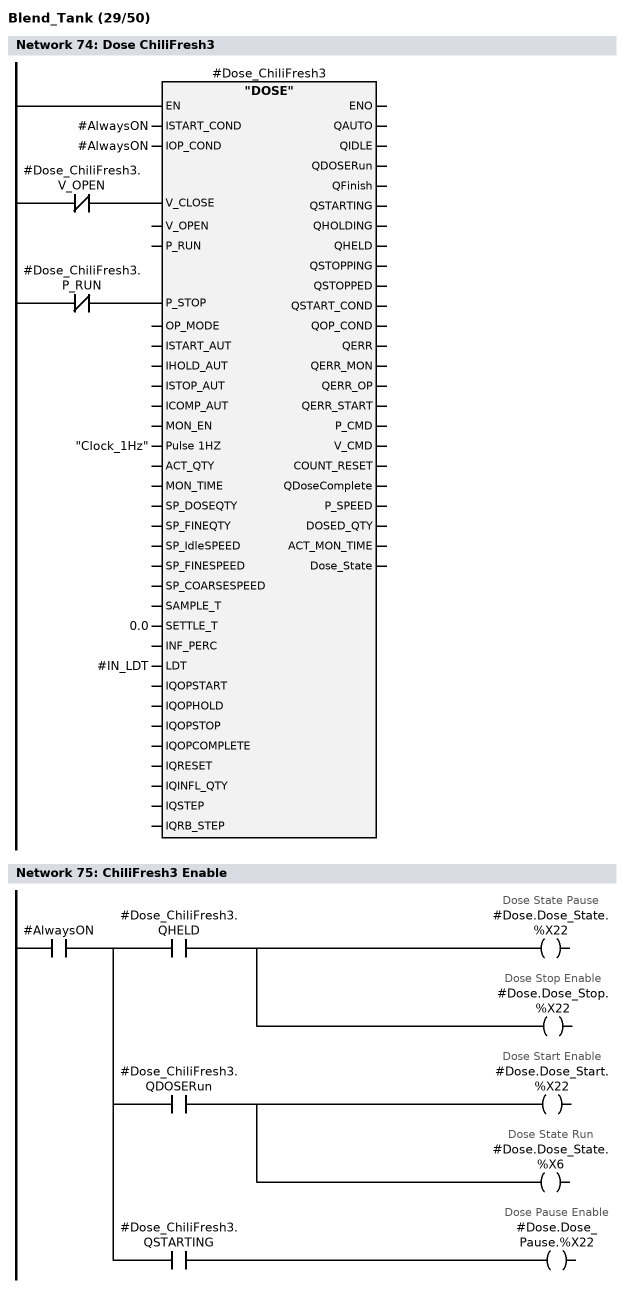
   RUNG wire#powerrail
      #Dose_ChiliFresh3(V_CLOSE := wire#w1, P_STOP := wire#w2, ISTART_COND := #AlwaysON, IOP_COND := #AlwaysON, V_OPEN :=, P_RUN :=, OP_MODE :=, ISTART_AUT :=, IHOLD_AUT :=, ISTOP_AUT :=, ICOMP_AUT :=, MON_EN :=, "Pulse 1HZ" := "Clock_1Hz", ACT_QTY :=, MON_TIME :=, SP_DOSEQTY :=, SP_FINEQTY :=, SP_IdleSPEED :=, SP_FINESPEED :=, SP_COARSESPEED :=, SAMPLE_T :=, SETTLE_T := 0.0, INF_PERC :=, LDT := #IN_LDT, IQOPSTART :=, IQOPHOLD :=, IQOPSTOP :=, IQOPCOMPLETE :=, IQRESET :=, IQINFL_QTY :=, IQSTEP :=, IQRB_STEP :=, QAUTO =>, QIDLE =>, QDOSERun =>, QFinish =>, QSTARTING =>, QHOLDING =>, QHELD =>, QSTOPPING =>, QSTOPPED =>, QSTART_COND =>, QOP_COND =>, QERR =>, QERR_MON =>, QERR_OP =>, QERR_START =>, P_CMD =>, V_CMD =>, COUNT_RESET =>, QDoseComplete =>, P_SPEED =>, DOSED_QTY =>, ACT_MON_TIME =>, Dose_State =>)
   END_RUNG
   RUNG wire#powerrail
      I_Contact( #Dose_ChiliFresh3.V_OPEN )
   END_RUNG wire#w1
   RUNG wire#powerrail
      I_Contact( #Dose_ChiliFresh3.P_RUN )
   END_RUNG wire#w2
   // the same network as SCL:
   #Dose_ChiliFresh3(ISTART_COND := #AlwaysON,   // "DOSE"
                     IOP_COND := #AlwaysON,
                     V_CLOSE := NOT #Dose_ChiliFresh3.V_OPEN,
                     P_STOP := NOT #Dose_ChiliFresh3.P_RUN,
                     "Pulse 1HZ" := "Clock_1Hz",
                     SETTLE_T := 0.0,
                     LDT := #IN_LDT);
END_REGION

REGION Network 75: ChiliFresh3 Enable
   RUNG wire#powerrail
      Contact( #AlwaysON )
      wire#w1
      Contact( #Dose_ChiliFresh3.QHELD )
      wire#w2
      Coil( #Dose.Dose_State.%X22 )   // Dose State Pause
   END_RUNG
   RUNG wire#w2
      Coil( #Dose.Dose_Stop.%X22 )   // Dose Stop Enable
   END_RUNG
   RUNG wire#w1
      Contact( #Dose_ChiliFresh3.QDOSERun )
      wire#w3
      Coil( #Dose.Dose_Start.%X22 )   // Dose Start Enable
   END_RUNG
   RUNG wire#w3
      Coil( #Dose.Dose_State.%X6 )   // Dose State Run
   END_RUNG
   RUNG wire#w1
      Contact( #Dose_ChiliFresh3.QSTARTING )
      Coil( #Dose.Dose_Pause.%X22 )   // Dose Pause Enable
   END_RUNG
   // the same network as SCL:
   #Dose.Dose_State.%X22 := #AlwaysON AND #Dose_ChiliFresh3.QHELD;   // Dose State Pause
   #Dose.Dose_Stop.%X22 := #Dose.Dose_State.%X22;   // Dose Stop Enable
   #Dose.Dose_Start.%X22 := #AlwaysON AND #Dose_ChiliFresh3.QDOSERun;   // Dose Start Enable
   #Dose.Dose_State.%X6 := #Dose.Dose_Start.%X22;   // Dose State Run
   #Dose.Dose_Pause.%X22 := #AlwaysON AND #Dose_ChiliFresh3.QSTARTING;   // Dose Pause Enable
END_REGION

REGION Network 76: ChiliFresh3 Header Req
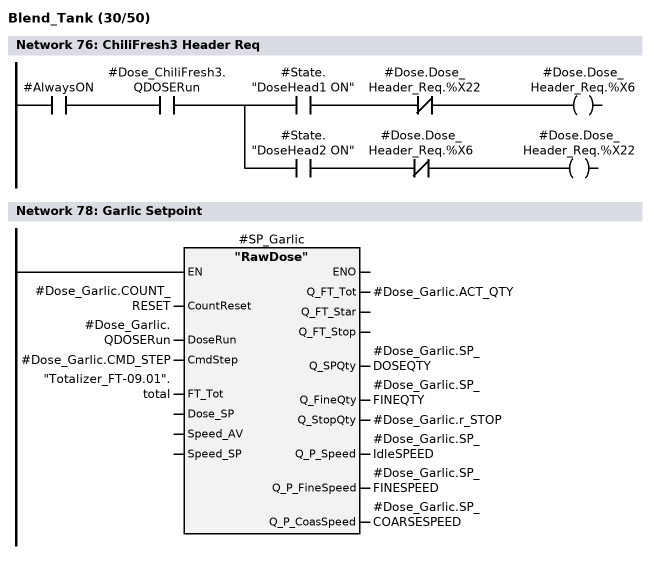
   RUNG wire#powerrail
      Contact( #AlwaysON )
      Contact( #Dose_ChiliFresh3.QDOSERun )
      wire#w1
      Contact( #State."DoseHead1 ON" )
      I_Contact( #Dose.Dose_Header_Req.%X22 )
      Coil( #Dose.Dose_Header_Req.%X6 )
   END_RUNG
   RUNG wire#w1
      Contact( #State."DoseHead2 ON" )
      I_Contact( #Dose.Dose_Header_Req.%X6 )
      Coil( #Dose.Dose_Header_Req.%X22 )
   END_RUNG
   // the same network as SCL:
   #_w1 := #AlwaysON AND #Dose_ChiliFresh3.QDOSERun;
   #Dose.Dose_Header_Req.%X6 := #_w1 AND #State."DoseHead1 ON" AND NOT #Dose.Dose_Header_Req.%X22;
   #Dose.Dose_Header_Req.%X22 := #_w1 AND #State."DoseHead2 ON" AND NOT #Dose.Dose_Header_Req.%X6;
END_REGION

REGION Network 78: Garlic Setpoint
   RUNG wire#powerrail
      #SP_Garlic(CountReset := #Dose_Garlic.COUNT_RESET, DoseRun := #Dose_Garlic.QDOSERun, CmdStep := #Dose_Garlic.CMD_STEP, FT_Tot := "Totalizer_FT-09.01".total, Dose_SP :=, Speed_AV :=, Speed_SP :=, Q_FT_Tot => #Dose_Garlic.ACT_QTY, Q_FT_Star =>, Q_FT_Stop =>, Q_SPQty => #Dose_Garlic.SP_DOSEQTY, Q_FineQty => #Dose_Garlic.SP_FINEQTY, Q_StopQty => #Dose_Garlic.r_STOP, Q_P_Speed => #Dose_Garlic.SP_IdleSPEED, Q_P_FineSpeed => #Dose_Garlic.SP_FINESPEED, Q_P_CoasSpeed => #Dose_Garlic.SP_COARSESPEED)
   END_RUNG
   // the same network as SCL:
   #SP_Garlic(CountReset := #Dose_Garlic.COUNT_RESET,   // "RawDose"
              DoseRun := #Dose_Garlic.QDOSERun,
              CmdStep := #Dose_Garlic.CMD_STEP,
              FT_Tot := "Totalizer_FT-09.01".total,
              Q_FT_Tot => #Dose_Garlic.ACT_QTY,
              Q_SPQty => #Dose_Garlic.SP_DOSEQTY,
              Q_FineQty => #Dose_Garlic.SP_FINEQTY,
              Q_StopQty => #Dose_Garlic.r_STOP,
              Q_P_Speed => #Dose_Garlic.SP_IdleSPEED,
              Q_P_FineSpeed => #Dose_Garlic.SP_FINESPEED,
              Q_P_CoasSpeed => #Dose_Garlic.SP_COARSESPEED);
END_REGION

REGION Network 79: Command Dose Garlic
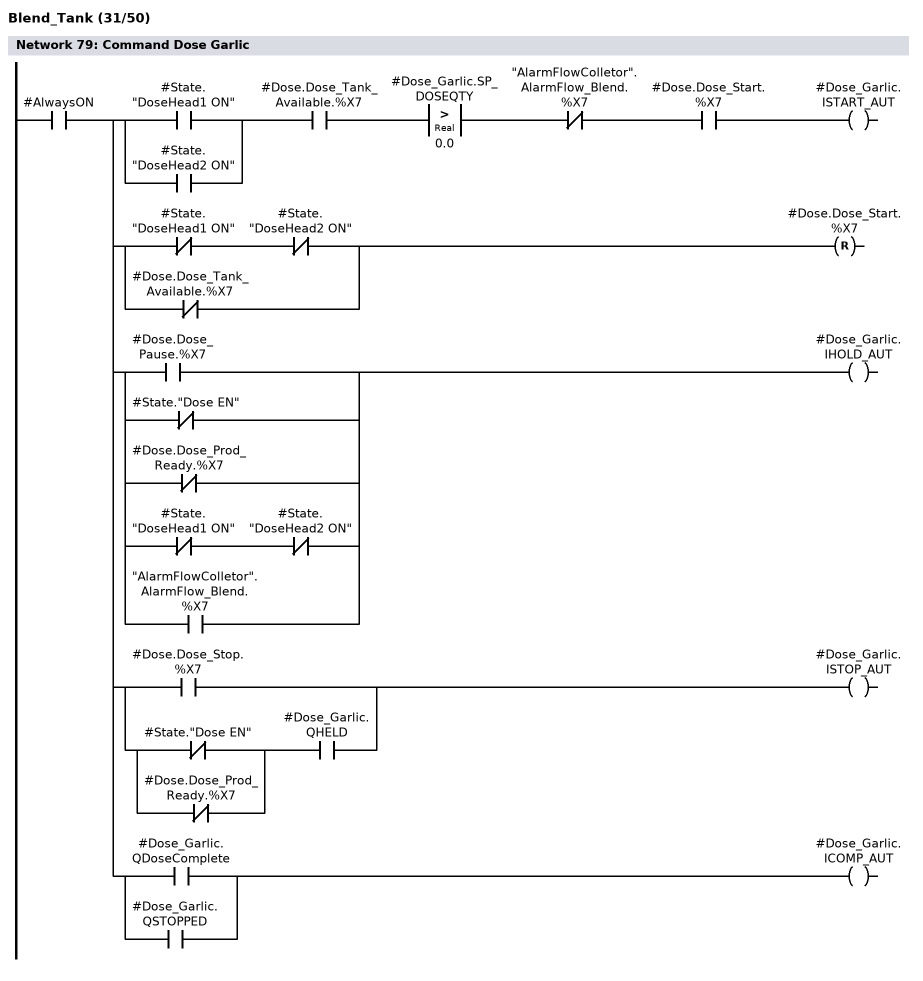
   RUNG wire#powerrail
      Contact( #AlwaysON )
      wire#w1
      Contact( #State."DoseHead1 ON" )
      wire#w2
      Contact( #Dose.Dose_Tank_Available.%X7 )
      { S7_Templates := "SrcType := Real" } GT_Contact(in1 := #Dose_Garlic.SP_DOSEQTY, in2 := 0.0)
      I_Contact( "AlarmFlowColletor".AlarmFlow_Blend.%X7 )
      Contact( #Dose.Dose_Start.%X7 )
      Coil( #Dose_Garlic.ISTART_AUT )
   END_RUNG
   RUNG wire#w1
      Contact( #State."DoseHead2 ON" )
   END_RUNG wire#w2
   RUNG wire#w1
      I_Contact( #State."DoseHead1 ON" )
      I_Contact( #State."DoseHead2 ON" )
      wire#w3
      R_Coil( #Dose.Dose_Start.%X7 )
   END_RUNG
   RUNG wire#w1
      I_Contact( #Dose.Dose_Tank_Available.%X7 )
   END_RUNG wire#w3
   RUNG wire#w1
      Contact( #Dose.Dose_Pause.%X7 )
      wire#w4
      Coil( #Dose_Garlic.IHOLD_AUT )
   END_RUNG
   RUNG wire#w1
      I_Contact( #State."Dose EN" )
   END_RUNG wire#w4
   RUNG wire#w1
      I_Contact( #Dose.Dose_Prod_Ready.%X7 )
   END_RUNG wire#w4
   RUNG wire#w1
      I_Contact( #State."DoseHead1 ON" )
      I_Contact( #State."DoseHead2 ON" )
   END_RUNG wire#w4
   RUNG wire#w1
      Contact( "AlarmFlowColletor".AlarmFlow_Blend.%X7 )
   END_RUNG wire#w4
   RUNG wire#w1
      Contact( #Dose.Dose_Stop.%X7 )
      wire#w5
      Coil( #Dose_Garlic.ISTOP_AUT )
   END_RUNG
   RUNG wire#w1
      I_Contact( #State."Dose EN" )
      wire#w6
      Contact( #Dose_Garlic.QHELD )
   END_RUNG wire#w5
   RUNG wire#w1
      I_Contact( #Dose.Dose_Prod_Ready.%X7 )
   END_RUNG wire#w6
   RUNG wire#w1
      Contact( #Dose_Garlic.QDoseComplete )
      wire#w7
      Coil( #Dose_Garlic.ICOMP_AUT )
   END_RUNG
   RUNG wire#w1
      Contact( #Dose_Garlic.QSTOPPED )
   END_RUNG wire#w7
   // the same network as SCL:
   #Dose_Garlic.ISTART_AUT := #AlwaysON AND (#State."DoseHead1 ON" OR #State."DoseHead2 ON") AND #Dose.Dose_Tank_Available.%X7 AND (#Dose_Garlic.SP_DOSEQTY > 0.0) AND NOT "AlarmFlowColletor".AlarmFlow_Blend.%X7 AND #Dose.Dose_Start.%X7;
   IF #AlwaysON AND ((NOT #State."DoseHead1 ON" AND NOT #State."DoseHead2 ON") OR NOT #Dose.Dose_Tank_Available.%X7) THEN
       #Dose.Dose_Start.%X7 := FALSE;
   END_IF;
   #Dose_Garlic.IHOLD_AUT := #AlwaysON AND (#Dose.Dose_Pause.%X7 OR NOT #State."Dose EN" OR NOT #Dose.Dose_Prod_Ready.%X7 OR (NOT #State."DoseHead1 ON" AND NOT #State."DoseHead2 ON") OR "AlarmFlowColletor".AlarmFlow_Blend.%X7);
   #Dose_Garlic.ISTOP_AUT := #AlwaysON AND (#Dose.Dose_Stop.%X7 OR ((NOT #State."Dose EN" OR NOT #Dose.Dose_Prod_Ready.%X7) AND #Dose_Garlic.QHELD));
   #Dose_Garlic.ICOMP_AUT := #AlwaysON AND (#Dose_Garlic.QDoseComplete OR #Dose_Garlic.QSTOPPED);
END_REGION

REGION Network 80: Dose Garlic
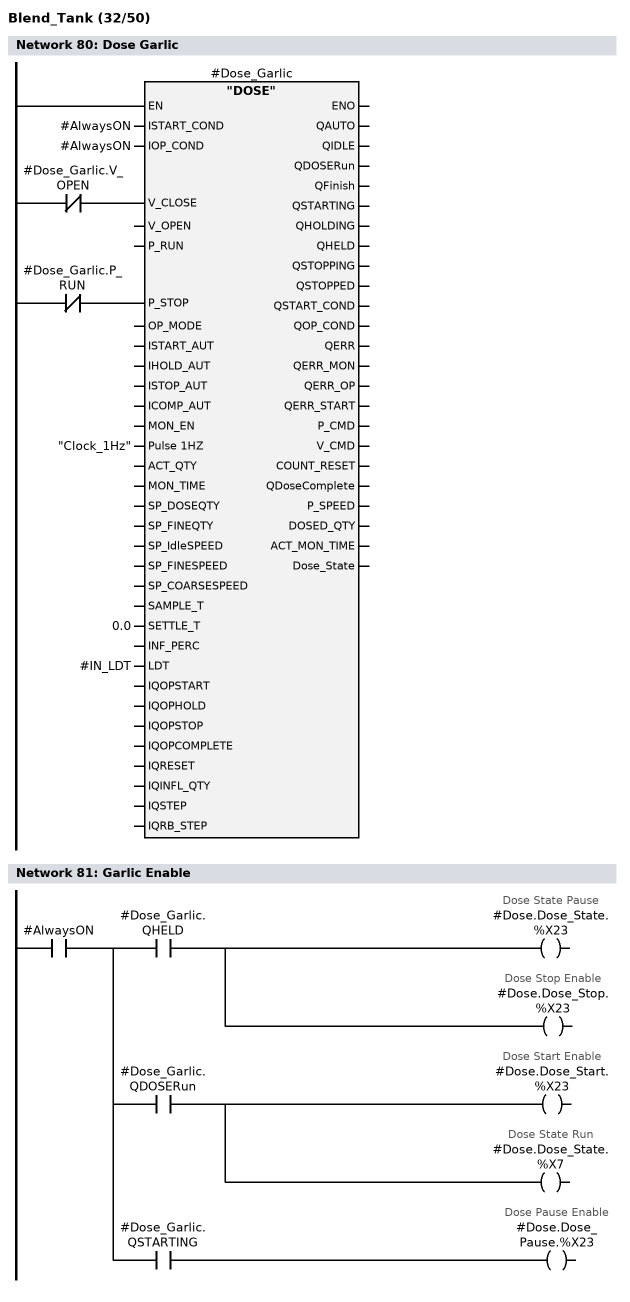
   RUNG wire#powerrail
      #Dose_Garlic(V_CLOSE := wire#w1, P_STOP := wire#w2, ISTART_COND := #AlwaysON, IOP_COND := #AlwaysON, V_OPEN :=, P_RUN :=, OP_MODE :=, ISTART_AUT :=, IHOLD_AUT :=, ISTOP_AUT :=, ICOMP_AUT :=, MON_EN :=, "Pulse 1HZ" := "Clock_1Hz", ACT_QTY :=, MON_TIME :=, SP_DOSEQTY :=, SP_FINEQTY :=, SP_IdleSPEED :=, SP_FINESPEED :=, SP_COARSESPEED :=, SAMPLE_T :=, SETTLE_T := 0.0, INF_PERC :=, LDT := #IN_LDT, IQOPSTART :=, IQOPHOLD :=, IQOPSTOP :=, IQOPCOMPLETE :=, IQRESET :=, IQINFL_QTY :=, IQSTEP :=, IQRB_STEP :=, QAUTO =>, QIDLE =>, QDOSERun =>, QFinish =>, QSTARTING =>, QHOLDING =>, QHELD =>, QSTOPPING =>, QSTOPPED =>, QSTART_COND =>, QOP_COND =>, QERR =>, QERR_MON =>, QERR_OP =>, QERR_START =>, P_CMD =>, V_CMD =>, COUNT_RESET =>, QDoseComplete =>, P_SPEED =>, DOSED_QTY =>, ACT_MON_TIME =>, Dose_State =>)
   END_RUNG
   RUNG wire#powerrail
      I_Contact( #Dose_Garlic.V_OPEN )
   END_RUNG wire#w1
   RUNG wire#powerrail
      I_Contact( #Dose_Garlic.P_RUN )
   END_RUNG wire#w2
   // the same network as SCL:
   #Dose_Garlic(ISTART_COND := #AlwaysON,   // "DOSE"
                IOP_COND := #AlwaysON,
                V_CLOSE := NOT #Dose_Garlic.V_OPEN,
                P_STOP := NOT #Dose_Garlic.P_RUN,
                "Pulse 1HZ" := "Clock_1Hz",
                SETTLE_T := 0.0,
                LDT := #IN_LDT);
END_REGION

REGION Network 81: Garlic Enable
   RUNG wire#powerrail
      Contact( #AlwaysON )
      wire#w1
      Contact( #Dose_Garlic.QHELD )
      wire#w2
      Coil( #Dose.Dose_State.%X23 )   // Dose State Pause
   END_RUNG
   RUNG wire#w2
      Coil( #Dose.Dose_Stop.%X23 )   // Dose Stop Enable
   END_RUNG
   RUNG wire#w1
      Contact( #Dose_Garlic.QDOSERun )
      wire#w3
      Coil( #Dose.Dose_Start.%X23 )   // Dose Start Enable
   END_RUNG
   RUNG wire#w3
      Coil( #Dose.Dose_State.%X7 )   // Dose State Run
   END_RUNG
   RUNG wire#w1
      Contact( #Dose_Garlic.QSTARTING )
      Coil( #Dose.Dose_Pause.%X23 )   // Dose Pause Enable
   END_RUNG
   // the same network as SCL:
   #Dose.Dose_State.%X23 := #AlwaysON AND #Dose_Garlic.QHELD;   // Dose State Pause
   #Dose.Dose_Stop.%X23 := #Dose.Dose_State.%X23;   // Dose Stop Enable
   #Dose.Dose_Start.%X23 := #AlwaysON AND #Dose_Garlic.QDOSERun;   // Dose Start Enable
   #Dose.Dose_State.%X7 := #Dose.Dose_Start.%X23;   // Dose State Run
   #Dose.Dose_Pause.%X23 := #AlwaysON AND #Dose_Garlic.QSTARTING;   // Dose Pause Enable
END_REGION

REGION Network 82: Garlic Header Req
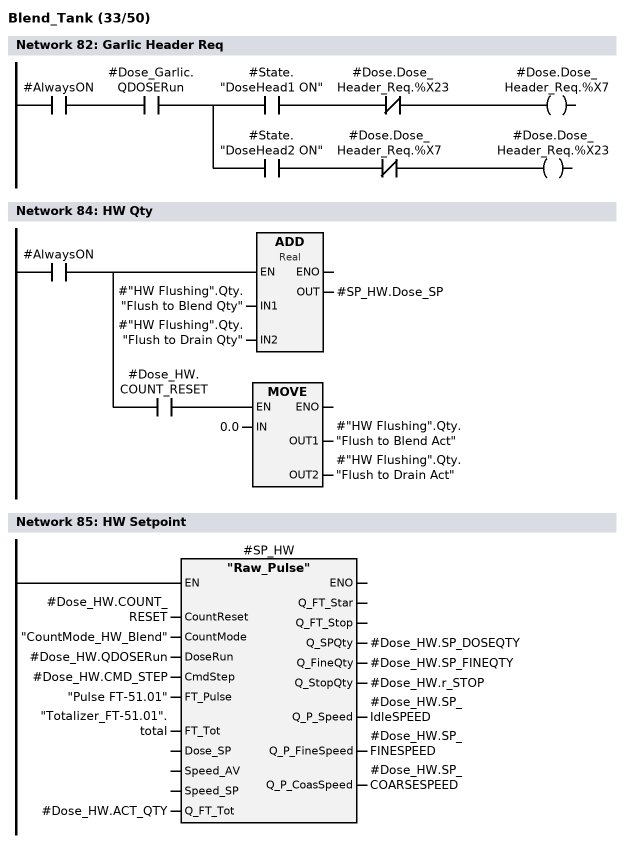
   RUNG wire#powerrail
      Contact( #AlwaysON )
      Contact( #Dose_Garlic.QDOSERun )
      wire#w1
      Contact( #State."DoseHead1 ON" )
      I_Contact( #Dose.Dose_Header_Req.%X23 )
      Coil( #Dose.Dose_Header_Req.%X7 )
   END_RUNG
   RUNG wire#w1
      Contact( #State."DoseHead2 ON" )
      I_Contact( #Dose.Dose_Header_Req.%X7 )
      Coil( #Dose.Dose_Header_Req.%X23 )
   END_RUNG
   // the same network as SCL:
   #_w1 := #AlwaysON AND #Dose_Garlic.QDOSERun;
   #Dose.Dose_Header_Req.%X7 := #_w1 AND #State."DoseHead1 ON" AND NOT #Dose.Dose_Header_Req.%X23;
   #Dose.Dose_Header_Req.%X23 := #_w1 AND #State."DoseHead2 ON" AND NOT #Dose.Dose_Header_Req.%X7;
END_REGION

REGION Network 84: HW Qty
   RUNG wire#powerrail
      Contact( #AlwaysON )
      wire#w1
      { S7_Templates := "SrcType := Real" } Add(in1 := #"HW Flushing".Qty."Flush to Blend Qty", in2 := #"HW Flushing".Qty."Flush to Drain Qty", out => #SP_HW.Dose_SP)
   END_RUNG
   RUNG wire#w1
      Contact( #Dose_HW.COUNT_RESET )
      Move(in := 0.0, out1 => #"HW Flushing".Qty."Flush to Blend Act", out2 => #"HW Flushing".Qty."Flush to Drain Act")
   END_RUNG
   // the same network as SCL:
   IF #AlwaysON THEN
       #SP_HW.Dose_SP := #"HW Flushing".Qty."Flush to Blend Qty" + #"HW Flushing".Qty."Flush to Drain Qty";
   END_IF;
   IF #AlwaysON AND #Dose_HW.COUNT_RESET THEN
       #"HW Flushing".Qty."Flush to Blend Act" := 0.0;
       #"HW Flushing".Qty."Flush to Drain Act" := 0.0;
   END_IF;
END_REGION

REGION Network 85: HW Setpoint
   RUNG wire#powerrail
      #SP_HW(CountReset := #Dose_HW.COUNT_RESET, CountMode := "CountMode_HW_Blend", DoseRun := #Dose_HW.QDOSERun, CmdStep := #Dose_HW.CMD_STEP, FT_Pulse := "Pulse FT-51.01", FT_Tot := "Totalizer_FT-51.01".total, Dose_SP :=, Speed_AV :=, Speed_SP :=, Q_FT_Tot := #Dose_HW.ACT_QTY, Q_FT_Star =>, Q_FT_Stop =>, Q_SPQty => #Dose_HW.SP_DOSEQTY, Q_FineQty => #Dose_HW.SP_FINEQTY, Q_StopQty => #Dose_HW.r_STOP, Q_P_Speed => #Dose_HW.SP_IdleSPEED, Q_P_FineSpeed => #Dose_HW.SP_FINESPEED, Q_P_CoasSpeed => #Dose_HW.SP_COARSESPEED)
   END_RUNG
   // the same network as SCL:
   #SP_HW(CountReset := #Dose_HW.COUNT_RESET,   // "Raw_Pulse"
          CountMode := "CountMode_HW_Blend",
          DoseRun := #Dose_HW.QDOSERun,
          CmdStep := #Dose_HW.CMD_STEP,
          FT_Pulse := "Pulse FT-51.01",
          FT_Tot := "Totalizer_FT-51.01".total,
          Q_FT_Tot := #Dose_HW.ACT_QTY,
          Q_SPQty => #Dose_HW.SP_DOSEQTY,
          Q_FineQty => #Dose_HW.SP_FINEQTY,
          Q_StopQty => #Dose_HW.r_STOP,
          Q_P_Speed => #Dose_HW.SP_IdleSPEED,
          Q_P_FineSpeed => #Dose_HW.SP_FINESPEED,
          Q_P_CoasSpeed => #Dose_HW.SP_COARSESPEED);
END_REGION

REGION Network 86: Command Dose HW
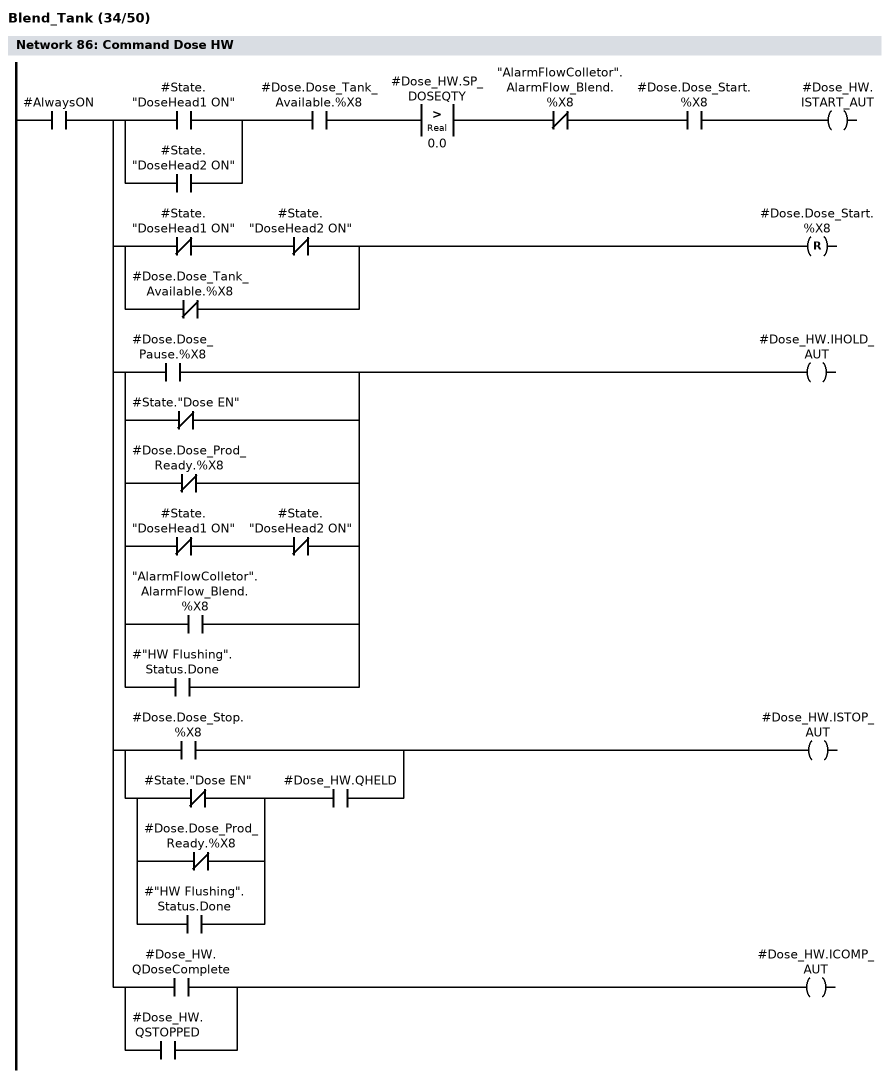
   RUNG wire#powerrail
      Contact( #AlwaysON )
      wire#w1
      Contact( #State."DoseHead1 ON" )
      wire#w2
      Contact( #Dose.Dose_Tank_Available.%X8 )
      { S7_Templates := "SrcType := Real" } GT_Contact(in1 := #Dose_HW.SP_DOSEQTY, in2 := 0.0)
      I_Contact( "AlarmFlowColletor".AlarmFlow_Blend.%X8 )
      Contact( #Dose.Dose_Start.%X8 )
      Coil( #Dose_HW.ISTART_AUT )
   END_RUNG
   RUNG wire#w1
      Contact( #State."DoseHead2 ON" )
   END_RUNG wire#w2
   RUNG wire#w1
      I_Contact( #State."DoseHead1 ON" )
      I_Contact( #State."DoseHead2 ON" )
      wire#w3
      R_Coil( #Dose.Dose_Start.%X8 )
   END_RUNG
   RUNG wire#w1
      I_Contact( #Dose.Dose_Tank_Available.%X8 )
   END_RUNG wire#w3
   RUNG wire#w1
      Contact( #Dose.Dose_Pause.%X8 )
      wire#w4
      Coil( #Dose_HW.IHOLD_AUT )
   END_RUNG
   RUNG wire#w1
      I_Contact( #State."Dose EN" )
   END_RUNG wire#w4
   RUNG wire#w1
      I_Contact( #Dose.Dose_Prod_Ready.%X8 )
   END_RUNG wire#w4
   RUNG wire#w1
      I_Contact( #State."DoseHead1 ON" )
      I_Contact( #State."DoseHead2 ON" )
   END_RUNG wire#w4
   RUNG wire#w1
      Contact( "AlarmFlowColletor".AlarmFlow_Blend.%X8 )
   END_RUNG wire#w4
   RUNG wire#w1
      Contact( #"HW Flushing".Status.Done )
   END_RUNG wire#w4
   RUNG wire#w1
      Contact( #Dose.Dose_Stop.%X8 )
      wire#w5
      Coil( #Dose_HW.ISTOP_AUT )
   END_RUNG
   RUNG wire#w1
      I_Contact( #State."Dose EN" )
      wire#w6
      Contact( #Dose_HW.QHELD )
   END_RUNG wire#w5
   RUNG wire#w1
      I_Contact( #Dose.Dose_Prod_Ready.%X8 )
   END_RUNG wire#w6
   RUNG wire#w1
      Contact( #"HW Flushing".Status.Done )
   END_RUNG wire#w6
   RUNG wire#w1
      Contact( #Dose_HW.QDoseComplete )
      wire#w7
      Coil( #Dose_HW.ICOMP_AUT )
   END_RUNG
   RUNG wire#w1
      Contact( #Dose_HW.QSTOPPED )
   END_RUNG wire#w7
   // the same network as SCL:
   #Dose_HW.ISTART_AUT := #AlwaysON AND (#State."DoseHead1 ON" OR #State."DoseHead2 ON") AND #Dose.Dose_Tank_Available.%X8 AND (#Dose_HW.SP_DOSEQTY > 0.0) AND NOT "AlarmFlowColletor".AlarmFlow_Blend.%X8 AND #Dose.Dose_Start.%X8;
   IF #AlwaysON AND ((NOT #State."DoseHead1 ON" AND NOT #State."DoseHead2 ON") OR NOT #Dose.Dose_Tank_Available.%X8) THEN
       #Dose.Dose_Start.%X8 := FALSE;
   END_IF;
   #Dose_HW.IHOLD_AUT := #AlwaysON AND (#Dose.Dose_Pause.%X8 OR NOT #State."Dose EN" OR NOT #Dose.Dose_Prod_Ready.%X8 OR (NOT #State."DoseHead1 ON" AND NOT #State."DoseHead2 ON") OR "AlarmFlowColletor".AlarmFlow_Blend.%X8 OR #"HW Flushing".Status.Done);
   #Dose_HW.ISTOP_AUT := #AlwaysON AND (#Dose.Dose_Stop.%X8 OR ((NOT #State."Dose EN" OR NOT #Dose.Dose_Prod_Ready.%X8 OR #"HW Flushing".Status.Done) AND #Dose_HW.QHELD));
   #Dose_HW.ICOMP_AUT := #AlwaysON AND (#Dose_HW.QDoseComplete OR #Dose_HW.QSTOPPED);
END_REGION

REGION Network 87: Dose HW
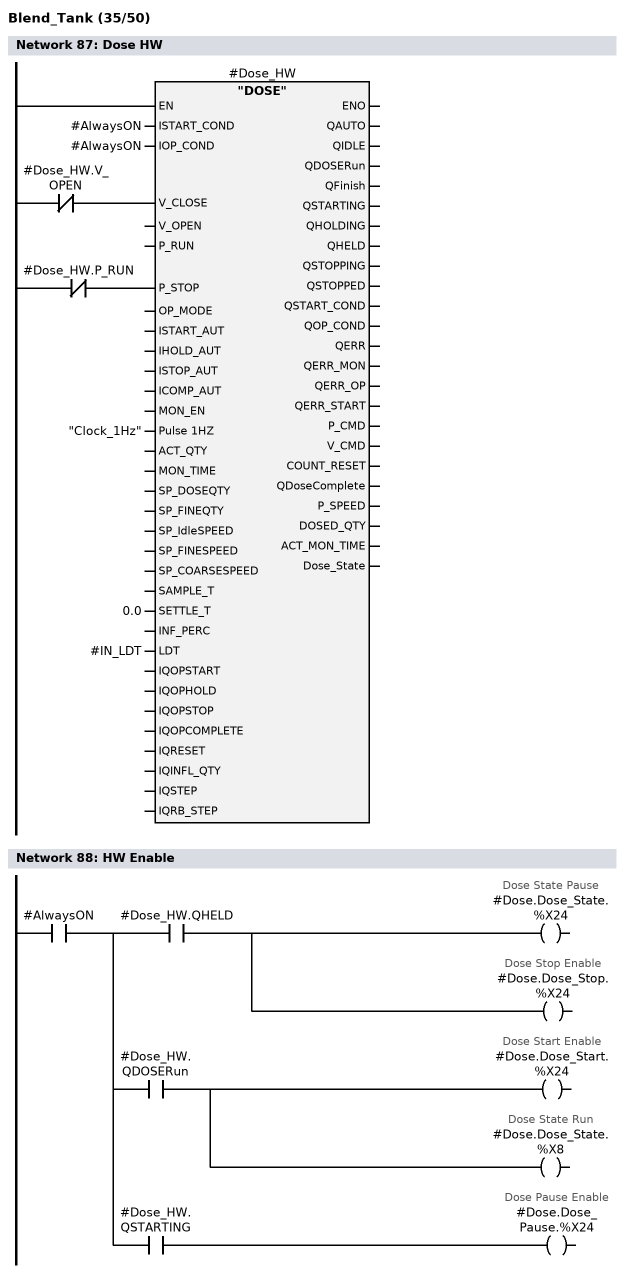
   RUNG wire#powerrail
      #Dose_HW(V_CLOSE := wire#w1, P_STOP := wire#w2, ISTART_COND := #AlwaysON, IOP_COND := #AlwaysON, V_OPEN :=, P_RUN :=, OP_MODE :=, ISTART_AUT :=, IHOLD_AUT :=, ISTOP_AUT :=, ICOMP_AUT :=, MON_EN :=, "Pulse 1HZ" := "Clock_1Hz", ACT_QTY :=, MON_TIME :=, SP_DOSEQTY :=, SP_FINEQTY :=, SP_IdleSPEED :=, SP_FINESPEED :=, SP_COARSESPEED :=, SAMPLE_T :=, SETTLE_T := 0.0, INF_PERC :=, LDT := #IN_LDT, IQOPSTART :=, IQOPHOLD :=, IQOPSTOP :=, IQOPCOMPLETE :=, IQRESET :=, IQINFL_QTY :=, IQSTEP :=, IQRB_STEP :=, QAUTO =>, QIDLE =>, QDOSERun =>, QFinish =>, QSTARTING =>, QHOLDING =>, QHELD =>, QSTOPPING =>, QSTOPPED =>, QSTART_COND =>, QOP_COND =>, QERR =>, QERR_MON =>, QERR_OP =>, QERR_START =>, P_CMD =>, V_CMD =>, COUNT_RESET =>, QDoseComplete =>, P_SPEED =>, DOSED_QTY =>, ACT_MON_TIME =>, Dose_State =>)
   END_RUNG
   RUNG wire#powerrail
      I_Contact( #Dose_HW.V_OPEN )
   END_RUNG wire#w1
   RUNG wire#powerrail
      I_Contact( #Dose_HW.P_RUN )
   END_RUNG wire#w2
   // the same network as SCL:
   #Dose_HW(ISTART_COND := #AlwaysON,   // "DOSE"
            IOP_COND := #AlwaysON,
            V_CLOSE := NOT #Dose_HW.V_OPEN,
            P_STOP := NOT #Dose_HW.P_RUN,
            "Pulse 1HZ" := "Clock_1Hz",
            SETTLE_T := 0.0,
            LDT := #IN_LDT);
END_REGION

REGION Network 88: HW Enable
   RUNG wire#powerrail
      Contact( #AlwaysON )
      wire#w1
      Contact( #Dose_HW.QHELD )
      wire#w2
      Coil( #Dose.Dose_State.%X24 )   // Dose State Pause
   END_RUNG
   RUNG wire#w2
      Coil( #Dose.Dose_Stop.%X24 )   // Dose Stop Enable
   END_RUNG
   RUNG wire#w1
      Contact( #Dose_HW.QDOSERun )
      wire#w3
      Coil( #Dose.Dose_Start.%X24 )   // Dose Start Enable
   END_RUNG
   RUNG wire#w3
      Coil( #Dose.Dose_State.%X8 )   // Dose State Run
   END_RUNG
   RUNG wire#w1
      Contact( #Dose_HW.QSTARTING )
      Coil( #Dose.Dose_Pause.%X24 )   // Dose Pause Enable
   END_RUNG
   // the same network as SCL:
   #Dose.Dose_State.%X24 := #AlwaysON AND #Dose_HW.QHELD;   // Dose State Pause
   #Dose.Dose_Stop.%X24 := #Dose.Dose_State.%X24;   // Dose Stop Enable
   #Dose.Dose_Start.%X24 := #AlwaysON AND #Dose_HW.QDOSERun;   // Dose Start Enable
   #Dose.Dose_State.%X8 := #Dose.Dose_Start.%X24;   // Dose State Run
   #Dose.Dose_Pause.%X24 := #AlwaysON AND #Dose_HW.QSTARTING;   // Dose Pause Enable
END_REGION

REGION Network 89: HW Header Req
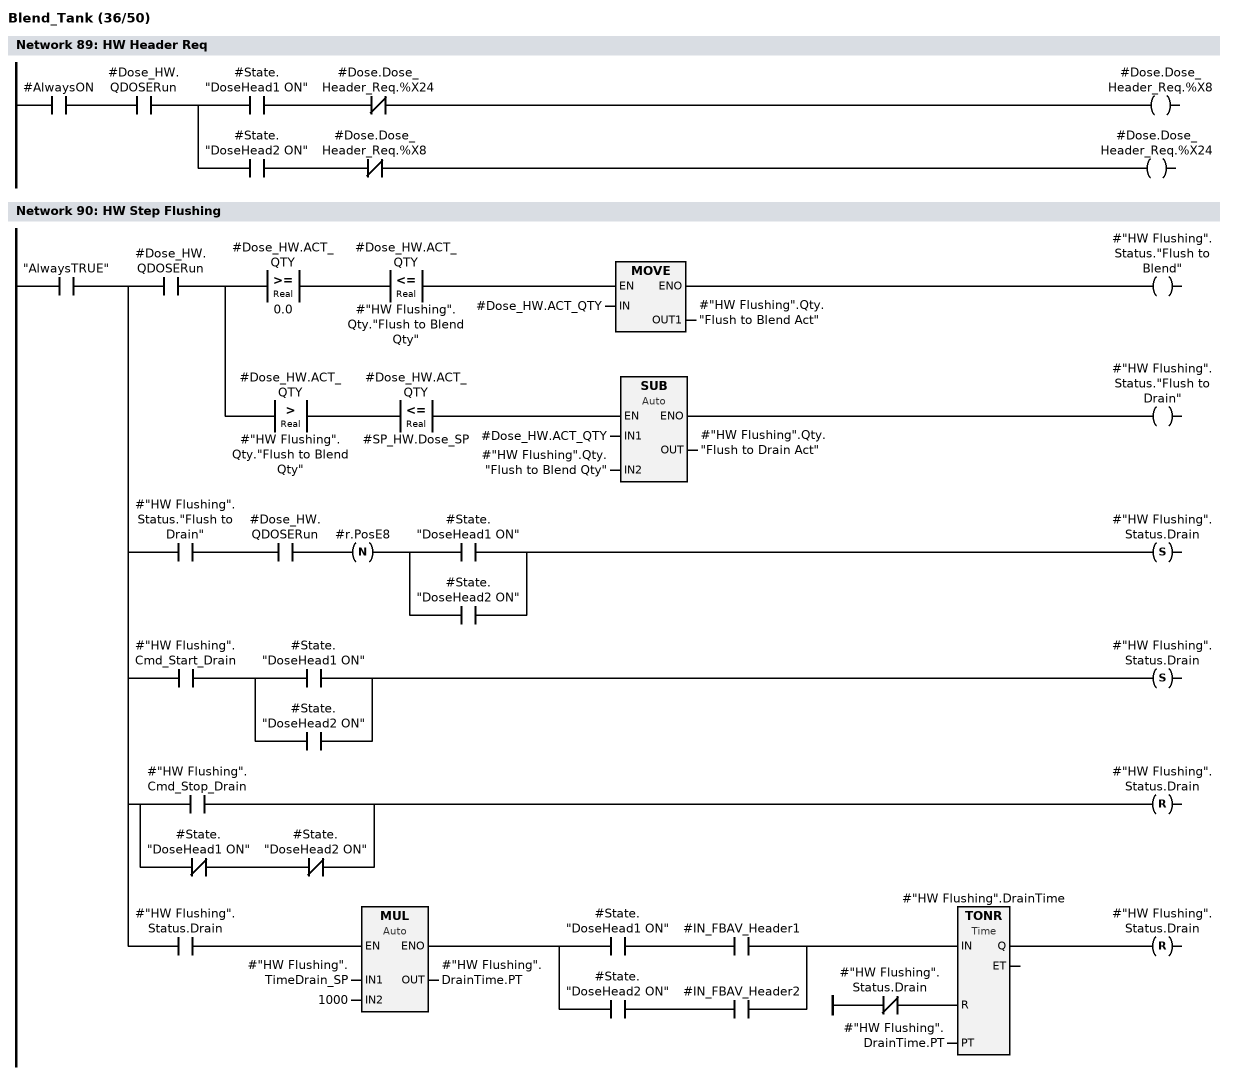
   RUNG wire#powerrail
      Contact( #AlwaysON )
      Contact( #Dose_HW.QDOSERun )
      wire#w1
      Contact( #State."DoseHead1 ON" )
      I_Contact( #Dose.Dose_Header_Req.%X24 )
      Coil( #Dose.Dose_Header_Req.%X8 )
   END_RUNG
   RUNG wire#w1
      Contact( #State."DoseHead2 ON" )
      I_Contact( #Dose.Dose_Header_Req.%X8 )
      Coil( #Dose.Dose_Header_Req.%X24 )
   END_RUNG
   // the same network as SCL:
   #_w1 := #AlwaysON AND #Dose_HW.QDOSERun;
   #Dose.Dose_Header_Req.%X8 := #_w1 AND #State."DoseHead1 ON" AND NOT #Dose.Dose_Header_Req.%X24;
   #Dose.Dose_Header_Req.%X24 := #_w1 AND #State."DoseHead2 ON" AND NOT #Dose.Dose_Header_Req.%X8;
END_REGION

REGION Network 90: HW Step Flushing
   RUNG wire#powerrail
      Contact( "AlwaysTRUE" )
      wire#w1
      Contact( #Dose_HW.QDOSERun )
      wire#w2
      { S7_Templates := "SrcType := Real" } GE_Contact(in1 := #Dose_HW.ACT_QTY, in2 := 0.0)
      { S7_Templates := "SrcType := Real" } LE_Contact(in1 := #Dose_HW.ACT_QTY, in2 := #"HW Flushing".Qty."Flush to Blend Qty")
      Move(in := #Dose_HW.ACT_QTY, out1 => #"HW Flushing".Qty."Flush to Blend Act")
      Coil( #"HW Flushing".Status."Flush to Blend" )
   END_RUNG
   RUNG wire#w2
      { S7_Templates := "SrcType := Real" } GT_Contact(in1 := #Dose_HW.ACT_QTY, in2 := #"HW Flushing".Qty."Flush to Blend Qty")
      { S7_Templates := "SrcType := Real" } LE_Contact(in1 := #Dose_HW.ACT_QTY, in2 := #SP_HW.Dose_SP)
      Sub(in1 := #Dose_HW.ACT_QTY, in2 := #"HW Flushing".Qty."Flush to Blend Qty", out => #"HW Flushing".Qty."Flush to Drain Act")
      Coil( #"HW Flushing".Status."Flush to Drain" )
   END_RUNG
   RUNG wire#w1
      Contact( #"HW Flushing".Status."Flush to Drain" )
      Contact( #Dose_HW.QDOSERun )
      N_Trig( #r.PosE8 )
      wire#w3
      Contact( #State."DoseHead1 ON" )
      wire#w4
      S_Coil( #"HW Flushing".Status.Drain )
   END_RUNG
   RUNG wire#w3
      Contact( #State."DoseHead2 ON" )
   END_RUNG wire#w4
   RUNG wire#w1
      Contact( #"HW Flushing".Cmd_Start_Drain )
      wire#w5
      Contact( #State."DoseHead1 ON" )
      wire#w6
      S_Coil( #"HW Flushing".Status.Drain )
   END_RUNG
   RUNG wire#w5
      Contact( #State."DoseHead2 ON" )
   END_RUNG wire#w6
   RUNG wire#w1
      Contact( #"HW Flushing".Cmd_Stop_Drain )
      wire#w7
      R_Coil( #"HW Flushing".Status.Drain )
   END_RUNG
   RUNG wire#w1
      I_Contact( #State."DoseHead1 ON" )
      I_Contact( #State."DoseHead2 ON" )
   END_RUNG wire#w7
   RUNG wire#w1
      Contact( #"HW Flushing".Status.Drain )
      Mul(in1 := #"HW Flushing".TimeDrain_SP, in2 := 1000, out => #"HW Flushing".DrainTime.PT)
      wire#w8
      Contact( #State."DoseHead1 ON" )
      Contact( #IN_FBAV_Header1 )
      wire#w9
      { S7_Templates := "time_type := Time" } #"HW Flushing".DrainTime.TONR(r := wire#w10, pt := #"HW Flushing".DrainTime.PT, et =>)
      R_Coil( #"HW Flushing".Status.Drain )
   END_RUNG
   RUNG wire#w8
      Contact( #State."DoseHead2 ON" )
      Contact( #IN_FBAV_Header2 )
   END_RUNG wire#w9
   RUNG wire#powerrail
      I_Contact( #"HW Flushing".Status.Drain )
   END_RUNG wire#w10
   // the same network as SCL:
   #_w1 := "AlwaysTRUE" AND #Dose_HW.QDOSERun;
   #_w2 := #_w1 AND (#Dose_HW.ACT_QTY >= 0.0) AND (#Dose_HW.ACT_QTY <= #"HW Flushing".Qty."Flush to Blend Qty");
   IF #_w2 THEN #"HW Flushing".Qty."Flush to Blend Act" := #Dose_HW.ACT_QTY; END_IF;
   #"HW Flushing".Status."Flush to Blend" := #_w2;
   #_w3 := #_w1 AND (#Dose_HW.ACT_QTY > #"HW Flushing".Qty."Flush to Blend Qty") AND (#Dose_HW.ACT_QTY <= #SP_HW.Dose_SP);
   IF #_w3 THEN
       #"HW Flushing".Qty."Flush to Drain Act" := #Dose_HW.ACT_QTY - #"HW Flushing".Qty."Flush to Blend Qty";
   END_IF;
   #"HW Flushing".Status."Flush to Drain" := #_w3;
   #_w4 := "AlwaysTRUE" AND #"HW Flushing".Status."Flush to Drain" AND #Dose_HW.QDOSERun;
   #_w5 := NOT #_w4 AND #r.PosE8;   // falling edge
   #r.PosE8 := #_w4;
   IF #_w5 AND (#State."DoseHead1 ON" OR #State."DoseHead2 ON") THEN
       #"HW Flushing".Status.Drain := TRUE;
   END_IF;
   IF "AlwaysTRUE" AND #"HW Flushing".Cmd_Start_Drain AND (#State."DoseHead1 ON" OR #State."DoseHead2 ON") THEN
       #"HW Flushing".Status.Drain := TRUE;
   END_IF;
   IF "AlwaysTRUE" AND (#"HW Flushing".Cmd_Stop_Drain OR (NOT #State."DoseHead1 ON" AND NOT #State."DoseHead2 ON")) THEN
       #"HW Flushing".Status.Drain := FALSE;
   END_IF;
   #_w6 := "AlwaysTRUE" AND #"HW Flushing".Status.Drain;
   IF #_w6 THEN #"HW Flushing".DrainTime.PT := #"HW Flushing".TimeDrain_SP * 1000; END_IF;
   #"HW Flushing".DrainTime.TONR(IN := #_w6 AND ((#State."DoseHead1 ON" AND #IN_FBAV_Header1) OR (#State."DoseHead2 ON" AND #IN_FBAV_Header2)),
                           R := NOT #"HW Flushing".Status.Drain,
                           PT := #"HW Flushing".DrainTime.PT);
   IF #"HW Flushing".DrainTime.Q THEN #"HW Flushing".Status.Drain := FALSE; END_IF;
END_REGION

REGION Network 92: Vinegar Setpoint
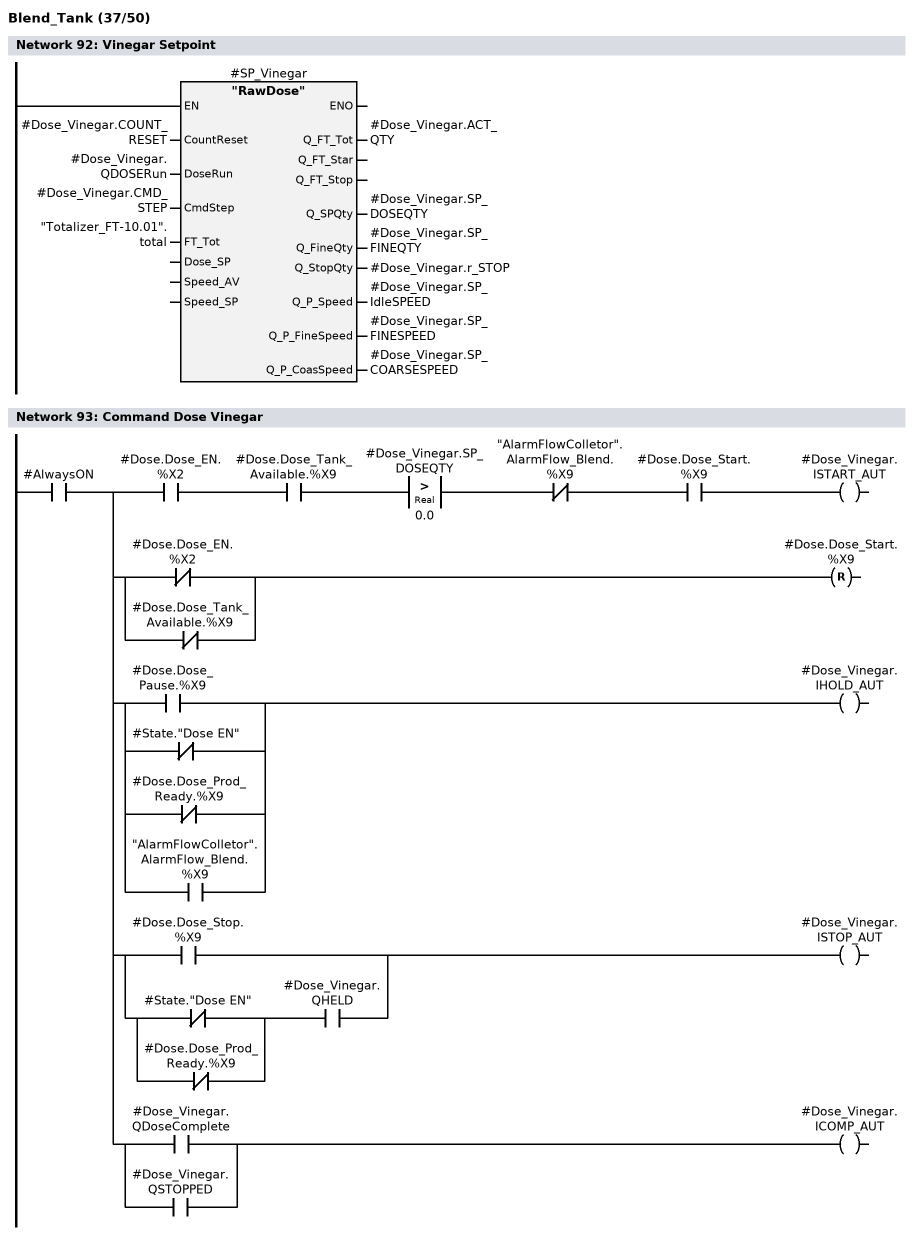
   RUNG wire#powerrail
      #SP_Vinegar(CountReset := #Dose_Vinegar.COUNT_RESET, DoseRun := #Dose_Vinegar.QDOSERun, CmdStep := #Dose_Vinegar.CMD_STEP, FT_Tot := "Totalizer_FT-10.01".total, Dose_SP :=, Speed_AV :=, Speed_SP :=, Q_FT_Tot => #Dose_Vinegar.ACT_QTY, Q_FT_Star =>, Q_FT_Stop =>, Q_SPQty => #Dose_Vinegar.SP_DOSEQTY, Q_FineQty => #Dose_Vinegar.SP_FINEQTY, Q_StopQty => #Dose_Vinegar.r_STOP, Q_P_Speed => #Dose_Vinegar.SP_IdleSPEED, Q_P_FineSpeed => #Dose_Vinegar.SP_FINESPEED, Q_P_CoasSpeed => #Dose_Vinegar.SP_COARSESPEED)
   END_RUNG
   // the same network as SCL:
   #SP_Vinegar(CountReset := #Dose_Vinegar.COUNT_RESET,   // "RawDose"
               DoseRun := #Dose_Vinegar.QDOSERun,
               CmdStep := #Dose_Vinegar.CMD_STEP,
               FT_Tot := "Totalizer_FT-10.01".total,
               Q_FT_Tot => #Dose_Vinegar.ACT_QTY,
               Q_SPQty => #Dose_Vinegar.SP_DOSEQTY,
               Q_FineQty => #Dose_Vinegar.SP_FINEQTY,
               Q_StopQty => #Dose_Vinegar.r_STOP,
               Q_P_Speed => #Dose_Vinegar.SP_IdleSPEED,
               Q_P_FineSpeed => #Dose_Vinegar.SP_FINESPEED,
               Q_P_CoasSpeed => #Dose_Vinegar.SP_COARSESPEED);
END_REGION

REGION Network 93: Command Dose Vinegar
   RUNG wire#powerrail
      Contact( #AlwaysON )
      wire#w1
      Contact( #Dose.Dose_EN.%X2 )
      Contact( #Dose.Dose_Tank_Available.%X9 )
      { S7_Templates := "SrcType := Real" } GT_Contact(in1 := #Dose_Vinegar.SP_DOSEQTY, in2 := 0.0)
      I_Contact( "AlarmFlowColletor".AlarmFlow_Blend.%X9 )
      Contact( #Dose.Dose_Start.%X9 )
      Coil( #Dose_Vinegar.ISTART_AUT )
   END_RUNG
   RUNG wire#w1
      I_Contact( #Dose.Dose_EN.%X2 )
      wire#w2
      R_Coil( #Dose.Dose_Start.%X9 )
   END_RUNG
   RUNG wire#w1
      I_Contact( #Dose.Dose_Tank_Available.%X9 )
   END_RUNG wire#w2
   RUNG wire#w1
      Contact( #Dose.Dose_Pause.%X9 )
      wire#w3
      Coil( #Dose_Vinegar.IHOLD_AUT )
   END_RUNG
   RUNG wire#w1
      I_Contact( #State."Dose EN" )
   END_RUNG wire#w3
   RUNG wire#w1
      I_Contact( #Dose.Dose_Prod_Ready.%X9 )
   END_RUNG wire#w3
   RUNG wire#w1
      Contact( "AlarmFlowColletor".AlarmFlow_Blend.%X9 )
   END_RUNG wire#w3
   RUNG wire#w1
      Contact( #Dose.Dose_Stop.%X9 )
      wire#w4
      Coil( #Dose_Vinegar.ISTOP_AUT )
   END_RUNG
   RUNG wire#w1
      I_Contact( #State."Dose EN" )
      wire#w5
      Contact( #Dose_Vinegar.QHELD )
   END_RUNG wire#w4
   RUNG wire#w1
      I_Contact( #Dose.Dose_Prod_Ready.%X9 )
   END_RUNG wire#w5
   RUNG wire#w1
      Contact( #Dose_Vinegar.QDoseComplete )
      wire#w6
      Coil( #Dose_Vinegar.ICOMP_AUT )
   END_RUNG
   RUNG wire#w1
      Contact( #Dose_Vinegar.QSTOPPED )
   END_RUNG wire#w6
   // the same network as SCL:
   #Dose_Vinegar.ISTART_AUT := #AlwaysON AND #Dose.Dose_EN.%X2 AND #Dose.Dose_Tank_Available.%X9 AND (#Dose_Vinegar.SP_DOSEQTY > 0.0) AND NOT "AlarmFlowColletor".AlarmFlow_Blend.%X9 AND #Dose.Dose_Start.%X9;
   IF #AlwaysON AND (NOT #Dose.Dose_EN.%X2 OR NOT #Dose.Dose_Tank_Available.%X9) THEN
       #Dose.Dose_Start.%X9 := FALSE;
   END_IF;
   #Dose_Vinegar.IHOLD_AUT := #AlwaysON AND (#Dose.Dose_Pause.%X9 OR NOT #State."Dose EN" OR NOT #Dose.Dose_Prod_Ready.%X9 OR "AlarmFlowColletor".AlarmFlow_Blend.%X9);
   #Dose_Vinegar.ISTOP_AUT := #AlwaysON AND (#Dose.Dose_Stop.%X9 OR ((NOT #State."Dose EN" OR NOT #Dose.Dose_Prod_Ready.%X9) AND #Dose_Vinegar.QHELD));
   #Dose_Vinegar.ICOMP_AUT := #AlwaysON AND (#Dose_Vinegar.QDoseComplete OR #Dose_Vinegar.QSTOPPED);
END_REGION

REGION Network 94: Dose Vinegar
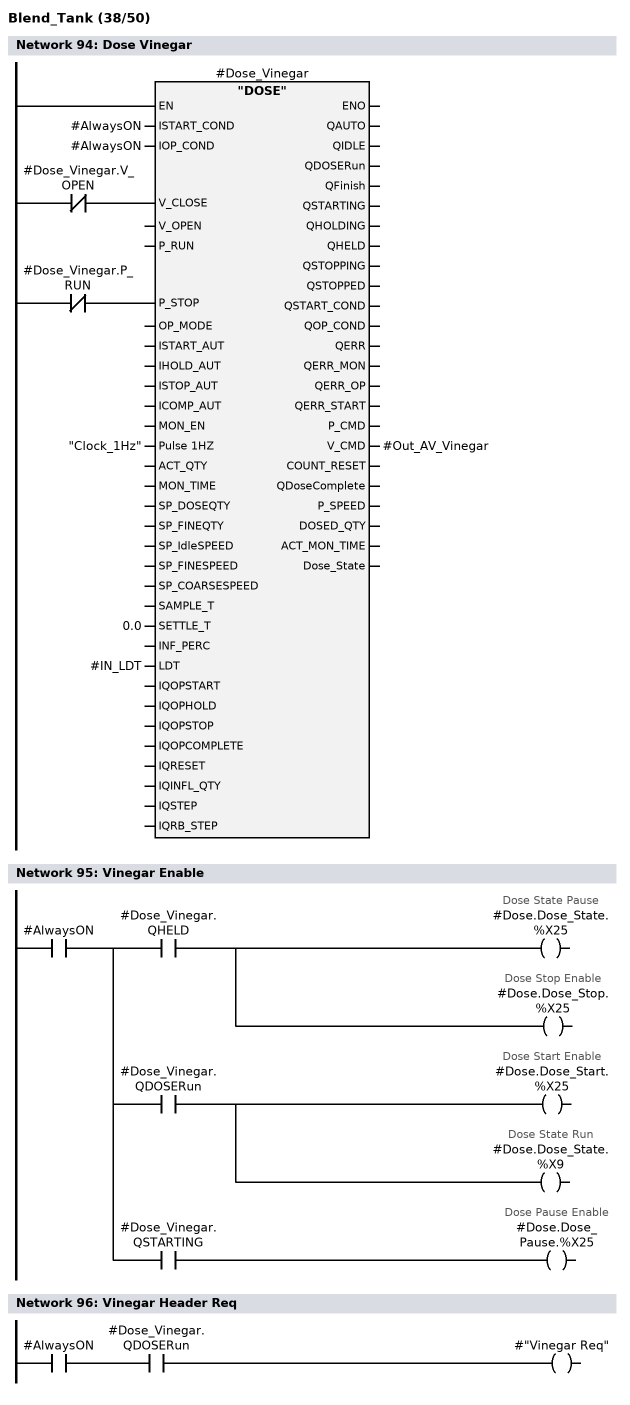
   RUNG wire#powerrail
      #Dose_Vinegar(V_CLOSE := wire#w1, P_STOP := wire#w2, ISTART_COND := #AlwaysON, IOP_COND := #AlwaysON, V_OPEN :=, P_RUN :=, OP_MODE :=, ISTART_AUT :=, IHOLD_AUT :=, ISTOP_AUT :=, ICOMP_AUT :=, MON_EN :=, "Pulse 1HZ" := "Clock_1Hz", ACT_QTY :=, MON_TIME :=, SP_DOSEQTY :=, SP_FINEQTY :=, SP_IdleSPEED :=, SP_FINESPEED :=, SP_COARSESPEED :=, SAMPLE_T :=, SETTLE_T := 0.0, INF_PERC :=, LDT := #IN_LDT, IQOPSTART :=, IQOPHOLD :=, IQOPSTOP :=, IQOPCOMPLETE :=, IQRESET :=, IQINFL_QTY :=, IQSTEP :=, IQRB_STEP :=, QAUTO =>, QIDLE =>, QDOSERun =>, QFinish =>, QSTARTING =>, QHOLDING =>, QHELD =>, QSTOPPING =>, QSTOPPED =>, QSTART_COND =>, QOP_COND =>, QERR =>, QERR_MON =>, QERR_OP =>, QERR_START =>, P_CMD =>, V_CMD => #Out_AV_Vinegar, COUNT_RESET =>, QDoseComplete =>, P_SPEED =>, DOSED_QTY =>, ACT_MON_TIME =>, Dose_State =>)
   END_RUNG
   RUNG wire#powerrail
      I_Contact( #Dose_Vinegar.V_OPEN )
   END_RUNG wire#w1
   RUNG wire#powerrail
      I_Contact( #Dose_Vinegar.P_RUN )
   END_RUNG wire#w2
   // the same network as SCL:
   #Dose_Vinegar(ISTART_COND := #AlwaysON,   // "DOSE"
                 IOP_COND := #AlwaysON,
                 V_CLOSE := NOT #Dose_Vinegar.V_OPEN,
                 P_STOP := NOT #Dose_Vinegar.P_RUN,
                 "Pulse 1HZ" := "Clock_1Hz",
                 SETTLE_T := 0.0,
                 LDT := #IN_LDT,
                 V_CMD => #Out_AV_Vinegar);
END_REGION

REGION Network 95: Vinegar Enable
   RUNG wire#powerrail
      Contact( #AlwaysON )
      wire#w1
      Contact( #Dose_Vinegar.QHELD )
      wire#w2
      Coil( #Dose.Dose_State.%X25 )   // Dose State Pause
   END_RUNG
   RUNG wire#w2
      Coil( #Dose.Dose_Stop.%X25 )   // Dose Stop Enable
   END_RUNG
   RUNG wire#w1
      Contact( #Dose_Vinegar.QDOSERun )
      wire#w3
      Coil( #Dose.Dose_Start.%X25 )   // Dose Start Enable
   END_RUNG
   RUNG wire#w3
      Coil( #Dose.Dose_State.%X9 )   // Dose State Run
   END_RUNG
   RUNG wire#w1
      Contact( #Dose_Vinegar.QSTARTING )
      Coil( #Dose.Dose_Pause.%X25 )   // Dose Pause Enable
   END_RUNG
   // the same network as SCL:
   #Dose.Dose_State.%X25 := #AlwaysON AND #Dose_Vinegar.QHELD;   // Dose State Pause
   #Dose.Dose_Stop.%X25 := #Dose.Dose_State.%X25;   // Dose Stop Enable
   #Dose.Dose_Start.%X25 := #AlwaysON AND #Dose_Vinegar.QDOSERun;   // Dose Start Enable
   #Dose.Dose_State.%X9 := #Dose.Dose_Start.%X25;   // Dose State Run
   #Dose.Dose_Pause.%X25 := #AlwaysON AND #Dose_Vinegar.QSTARTING;   // Dose Pause Enable
END_REGION

REGION Network 96: Vinegar Header Req
   RUNG wire#powerrail
      Contact( #AlwaysON )
      Contact( #Dose_Vinegar.QDOSERun )
      Coil( #"Vinegar Req" )
   END_RUNG
   // the same network as SCL:
   #"Vinegar Req" := #AlwaysON AND #Dose_Vinegar.QDOSERun;
END_REGION

REGION Network 98: Sugar Setpoint
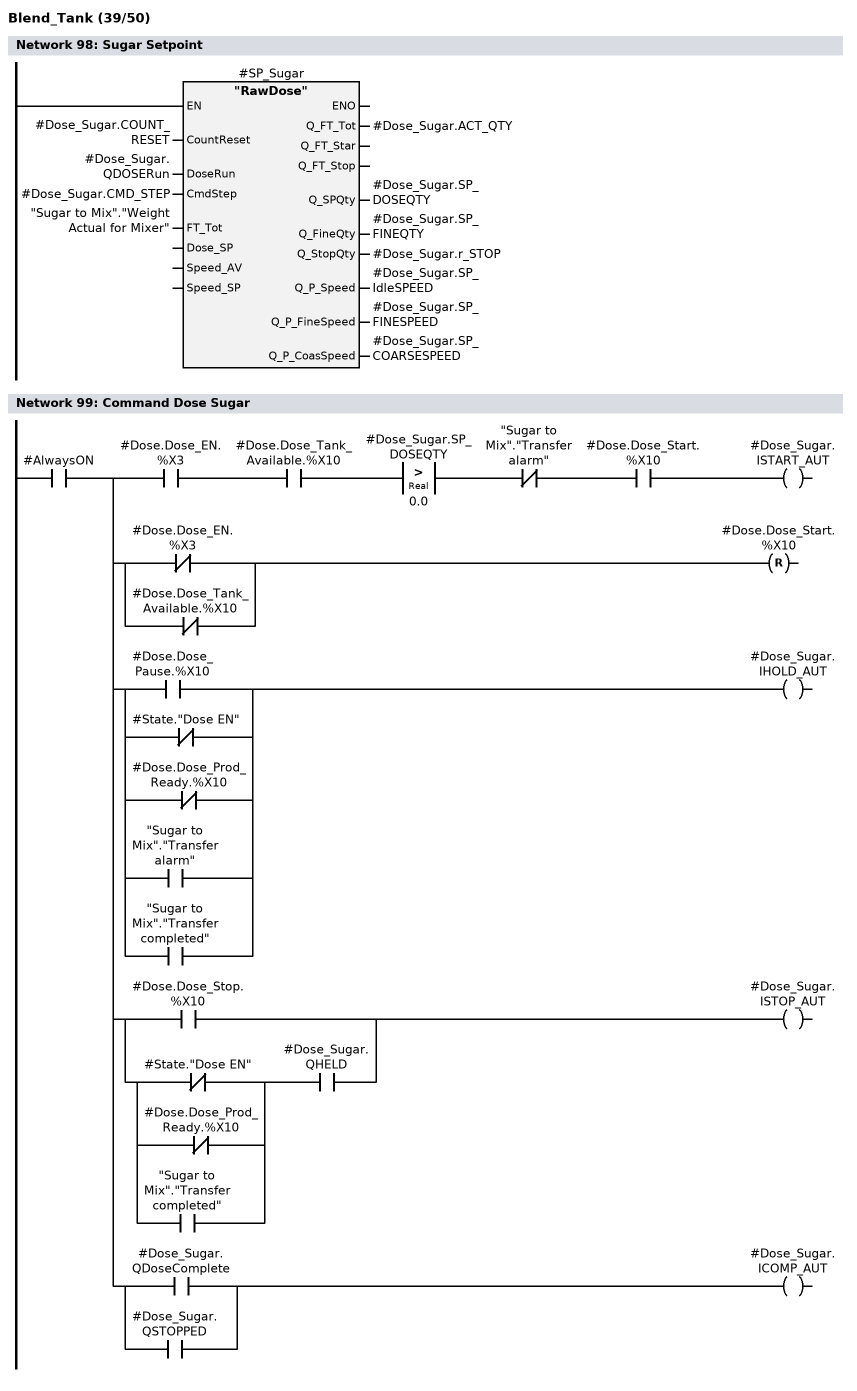
   RUNG wire#powerrail
      #SP_Sugar(CountReset := #Dose_Sugar.COUNT_RESET, DoseRun := #Dose_Sugar.QDOSERun, CmdStep := #Dose_Sugar.CMD_STEP, FT_Tot := "Sugar to Mix"."Weight Actual for Mixer", Dose_SP :=, Speed_AV :=, Speed_SP :=, Q_FT_Tot => #Dose_Sugar.ACT_QTY, Q_FT_Star =>, Q_FT_Stop =>, Q_SPQty => #Dose_Sugar.SP_DOSEQTY, Q_FineQty => #Dose_Sugar.SP_FINEQTY, Q_StopQty => #Dose_Sugar.r_STOP, Q_P_Speed => #Dose_Sugar.SP_IdleSPEED, Q_P_FineSpeed => #Dose_Sugar.SP_FINESPEED, Q_P_CoasSpeed => #Dose_Sugar.SP_COARSESPEED)
   END_RUNG
   // the same network as SCL:
   #SP_Sugar(CountReset := #Dose_Sugar.COUNT_RESET,   // "RawDose"
             DoseRun := #Dose_Sugar.QDOSERun,
             CmdStep := #Dose_Sugar.CMD_STEP,
             FT_Tot := "Sugar to Mix"."Weight Actual for Mixer",
             Q_FT_Tot => #Dose_Sugar.ACT_QTY,
             Q_SPQty => #Dose_Sugar.SP_DOSEQTY,
             Q_FineQty => #Dose_Sugar.SP_FINEQTY,
             Q_StopQty => #Dose_Sugar.r_STOP,
             Q_P_Speed => #Dose_Sugar.SP_IdleSPEED,
             Q_P_FineSpeed => #Dose_Sugar.SP_FINESPEED,
             Q_P_CoasSpeed => #Dose_Sugar.SP_COARSESPEED);
END_REGION

REGION Network 99: Command Dose Sugar
   RUNG wire#powerrail
      Contact( #AlwaysON )
      wire#w1
      Contact( #Dose.Dose_EN.%X3 )
      Contact( #Dose.Dose_Tank_Available.%X10 )
      { S7_Templates := "SrcType := Real" } GT_Contact(in1 := #Dose_Sugar.SP_DOSEQTY, in2 := 0.0)
      I_Contact( "Sugar to Mix"."Transfer alarm" )
      Contact( #Dose.Dose_Start.%X10 )
      Coil( #Dose_Sugar.ISTART_AUT )
   END_RUNG
   RUNG wire#w1
      I_Contact( #Dose.Dose_EN.%X3 )
      wire#w2
      R_Coil( #Dose.Dose_Start.%X10 )
   END_RUNG
   RUNG wire#w1
      I_Contact( #Dose.Dose_Tank_Available.%X10 )
   END_RUNG wire#w2
   RUNG wire#w1
      Contact( #Dose.Dose_Pause.%X10 )
      wire#w3
      Coil( #Dose_Sugar.IHOLD_AUT )
   END_RUNG
   RUNG wire#w1
      I_Contact( #State."Dose EN" )
   END_RUNG wire#w3
   RUNG wire#w1
      I_Contact( #Dose.Dose_Prod_Ready.%X10 )
   END_RUNG wire#w3
   RUNG wire#w1
      Contact( "Sugar to Mix"."Transfer alarm" )
   END_RUNG wire#w3
   RUNG wire#w1
      Contact( "Sugar to Mix"."Transfer completed" )
   END_RUNG wire#w3
   RUNG wire#w1
      Contact( #Dose.Dose_Stop.%X10 )
      wire#w4
      Coil( #Dose_Sugar.ISTOP_AUT )
   END_RUNG
   RUNG wire#w1
      I_Contact( #State."Dose EN" )
      wire#w5
      Contact( #Dose_Sugar.QHELD )
   END_RUNG wire#w4
   RUNG wire#w1
      I_Contact( #Dose.Dose_Prod_Ready.%X10 )
   END_RUNG wire#w5
   RUNG wire#w1
      Contact( "Sugar to Mix"."Transfer completed" )
   END_RUNG wire#w5
   RUNG wire#w1
      Contact( #Dose_Sugar.QDoseComplete )
      wire#w6
      Coil( #Dose_Sugar.ICOMP_AUT )
   END_RUNG
   RUNG wire#w1
      Contact( #Dose_Sugar.QSTOPPED )
   END_RUNG wire#w6
   // the same network as SCL:
   #Dose_Sugar.ISTART_AUT := #AlwaysON AND #Dose.Dose_EN.%X3 AND #Dose.Dose_Tank_Available.%X10 AND (#Dose_Sugar.SP_DOSEQTY > 0.0) AND NOT "Sugar to Mix"."Transfer alarm" AND #Dose.Dose_Start.%X10;
   IF #AlwaysON AND (NOT #Dose.Dose_EN.%X3 OR NOT #Dose.Dose_Tank_Available.%X10) THEN
       #Dose.Dose_Start.%X10 := FALSE;
   END_IF;
   #Dose_Sugar.IHOLD_AUT := #AlwaysON AND (#Dose.Dose_Pause.%X10 OR NOT #State."Dose EN" OR NOT #Dose.Dose_Prod_Ready.%X10 OR "Sugar to Mix"."Transfer alarm" OR "Sugar to Mix"."Transfer completed");
   #Dose_Sugar.ISTOP_AUT := #AlwaysON AND (#Dose.Dose_Stop.%X10 OR ((NOT #State."Dose EN" OR NOT #Dose.Dose_Prod_Ready.%X10 OR "Sugar to Mix"."Transfer completed") AND #Dose_Sugar.QHELD));
   #Dose_Sugar.ICOMP_AUT := #AlwaysON AND (#Dose_Sugar.QDoseComplete OR #Dose_Sugar.QSTOPPED);
END_REGION

REGION Network 100: Dose Sugar
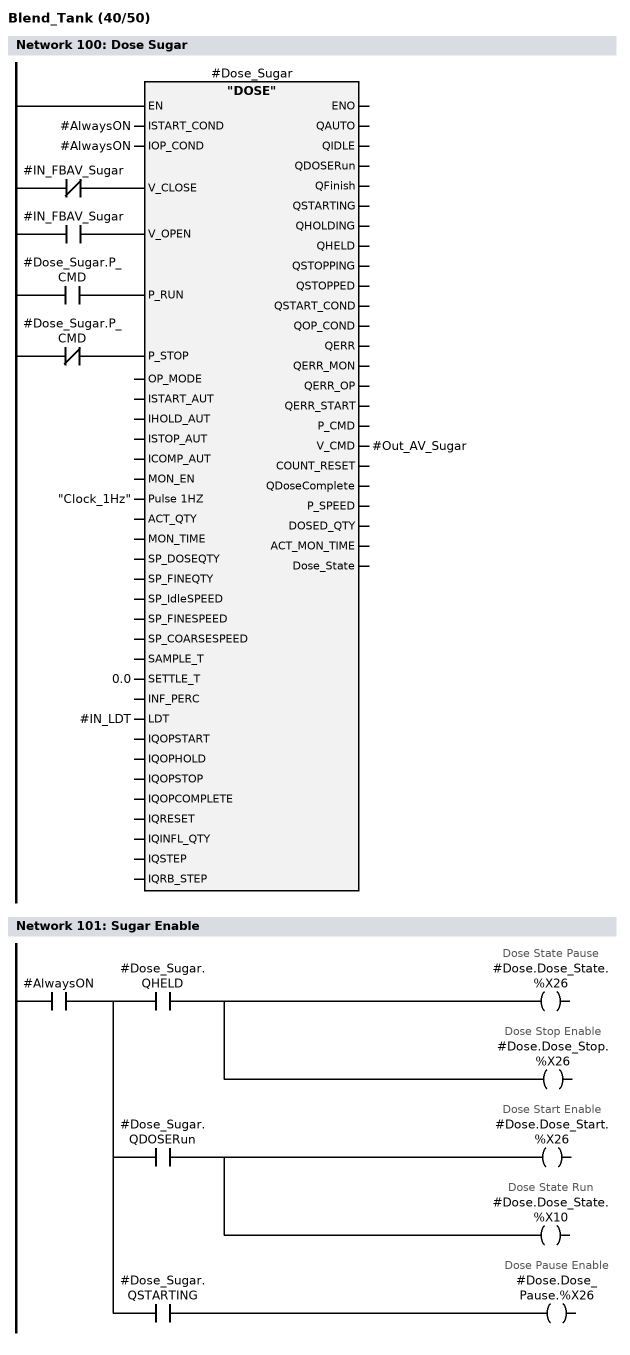
   RUNG wire#powerrail
      #Dose_Sugar(V_CLOSE := wire#w1, V_OPEN := wire#w2, P_RUN := wire#w3, P_STOP := wire#w4, ISTART_COND := #AlwaysON, IOP_COND := #AlwaysON, OP_MODE :=, ISTART_AUT :=, IHOLD_AUT :=, ISTOP_AUT :=, ICOMP_AUT :=, MON_EN :=, "Pulse 1HZ" := "Clock_1Hz", ACT_QTY :=, MON_TIME :=, SP_DOSEQTY :=, SP_FINEQTY :=, SP_IdleSPEED :=, SP_FINESPEED :=, SP_COARSESPEED :=, SAMPLE_T :=, SETTLE_T := 0.0, INF_PERC :=, LDT := #IN_LDT, IQOPSTART :=, IQOPHOLD :=, IQOPSTOP :=, IQOPCOMPLETE :=, IQRESET :=, IQINFL_QTY :=, IQSTEP :=, IQRB_STEP :=, QAUTO =>, QIDLE =>, QDOSERun =>, QFinish =>, QSTARTING =>, QHOLDING =>, QHELD =>, QSTOPPING =>, QSTOPPED =>, QSTART_COND =>, QOP_COND =>, QERR =>, QERR_MON =>, QERR_OP =>, QERR_START =>, P_CMD =>, V_CMD => #Out_AV_Sugar, COUNT_RESET =>, QDoseComplete =>, P_SPEED =>, DOSED_QTY =>, ACT_MON_TIME =>, Dose_State =>)
   END_RUNG
   RUNG wire#powerrail
      I_Contact( #IN_FBAV_Sugar )
   END_RUNG wire#w1
   RUNG wire#powerrail
      Contact( #IN_FBAV_Sugar )
   END_RUNG wire#w2
   RUNG wire#powerrail
      Contact( #Dose_Sugar.P_CMD )
   END_RUNG wire#w3
   RUNG wire#powerrail
      I_Contact( #Dose_Sugar.P_CMD )
   END_RUNG wire#w4
   // the same network as SCL:
   #Dose_Sugar(ISTART_COND := #AlwaysON,   // "DOSE"
               IOP_COND := #AlwaysON,
               V_CLOSE := NOT #IN_FBAV_Sugar,
               V_OPEN := #IN_FBAV_Sugar,
               P_RUN := #Dose_Sugar.P_CMD,
               P_STOP := NOT #Dose_Sugar.P_CMD,
               "Pulse 1HZ" := "Clock_1Hz",
               SETTLE_T := 0.0,
               LDT := #IN_LDT,
               V_CMD => #Out_AV_Sugar);
END_REGION

REGION Network 101: Sugar Enable
   RUNG wire#powerrail
      Contact( #AlwaysON )
      wire#w1
      Contact( #Dose_Sugar.QHELD )
      wire#w2
      Coil( #Dose.Dose_State.%X26 )   // Dose State Pause
   END_RUNG
   RUNG wire#w2
      Coil( #Dose.Dose_Stop.%X26 )   // Dose Stop Enable
   END_RUNG
   RUNG wire#w1
      Contact( #Dose_Sugar.QDOSERun )
      wire#w3
      Coil( #Dose.Dose_Start.%X26 )   // Dose Start Enable
   END_RUNG
   RUNG wire#w3
      Coil( #Dose.Dose_State.%X10 )   // Dose State Run
   END_RUNG
   RUNG wire#w1
      Contact( #Dose_Sugar.QSTARTING )
      Coil( #Dose.Dose_Pause.%X26 )   // Dose Pause Enable
   END_RUNG
   // the same network as SCL:
   #Dose.Dose_State.%X26 := #AlwaysON AND #Dose_Sugar.QHELD;   // Dose State Pause
   #Dose.Dose_Stop.%X26 := #Dose.Dose_State.%X26;   // Dose Stop Enable
   #Dose.Dose_Start.%X26 := #AlwaysON AND #Dose_Sugar.QDOSERun;   // Dose Start Enable
   #Dose.Dose_State.%X10 := #Dose.Dose_Start.%X26;   // Dose State Run
   #Dose.Dose_Pause.%X26 := #AlwaysON AND #Dose_Sugar.QSTARTING;   // Dose Pause Enable
END_REGION

REGION Network 102: Sugar Header Req
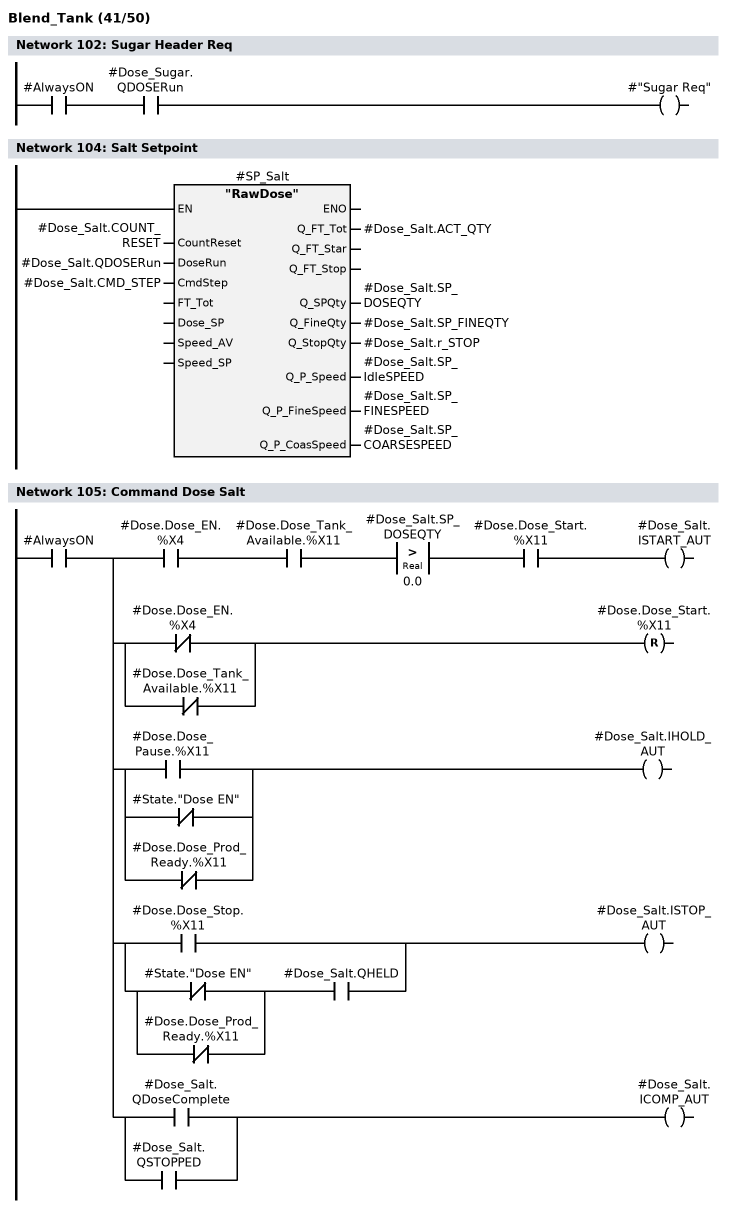
   RUNG wire#powerrail
      Contact( #AlwaysON )
      Contact( #Dose_Sugar.QDOSERun )
      Coil( #"Sugar Req" )
   END_RUNG
   // the same network as SCL:
   #"Sugar Req" := #AlwaysON AND #Dose_Sugar.QDOSERun;
END_REGION

REGION Network 104: Salt Setpoint
   RUNG wire#powerrail
      #SP_Salt(CountReset := #Dose_Salt.COUNT_RESET, DoseRun := #Dose_Salt.QDOSERun, CmdStep := #Dose_Salt.CMD_STEP, FT_Tot :=, Dose_SP :=, Speed_AV :=, Speed_SP :=, Q_FT_Tot => #Dose_Salt.ACT_QTY, Q_FT_Star =>, Q_FT_Stop =>, Q_SPQty => #Dose_Salt.SP_DOSEQTY, Q_FineQty => #Dose_Salt.SP_FINEQTY, Q_StopQty => #Dose_Salt.r_STOP, Q_P_Speed => #Dose_Salt.SP_IdleSPEED, Q_P_FineSpeed => #Dose_Salt.SP_FINESPEED, Q_P_CoasSpeed => #Dose_Salt.SP_COARSESPEED)
   END_RUNG
   // the same network as SCL:
   #SP_Salt(CountReset := #Dose_Salt.COUNT_RESET,   // "RawDose"
            DoseRun := #Dose_Salt.QDOSERun,
            CmdStep := #Dose_Salt.CMD_STEP,
            Q_FT_Tot => #Dose_Salt.ACT_QTY,
            Q_SPQty => #Dose_Salt.SP_DOSEQTY,
            Q_FineQty => #Dose_Salt.SP_FINEQTY,
            Q_StopQty => #Dose_Salt.r_STOP,
            Q_P_Speed => #Dose_Salt.SP_IdleSPEED,
            Q_P_FineSpeed => #Dose_Salt.SP_FINESPEED,
            Q_P_CoasSpeed => #Dose_Salt.SP_COARSESPEED);
END_REGION

REGION Network 105: Command Dose Salt
   RUNG wire#powerrail
      Contact( #AlwaysON )
      wire#w1
      Contact( #Dose.Dose_EN.%X4 )
      Contact( #Dose.Dose_Tank_Available.%X11 )
      { S7_Templates := "SrcType := Real" } GT_Contact(in1 := #Dose_Salt.SP_DOSEQTY, in2 := 0.0)
      Contact( #Dose.Dose_Start.%X11 )
      Coil( #Dose_Salt.ISTART_AUT )
   END_RUNG
   RUNG wire#w1
      I_Contact( #Dose.Dose_EN.%X4 )
      wire#w2
      R_Coil( #Dose.Dose_Start.%X11 )
   END_RUNG
   RUNG wire#w1
      I_Contact( #Dose.Dose_Tank_Available.%X11 )
   END_RUNG wire#w2
   RUNG wire#w1
      Contact( #Dose.Dose_Pause.%X11 )
      wire#w3
      Coil( #Dose_Salt.IHOLD_AUT )
   END_RUNG
   RUNG wire#w1
      I_Contact( #State."Dose EN" )
   END_RUNG wire#w3
   RUNG wire#w1
      I_Contact( #Dose.Dose_Prod_Ready.%X11 )
   END_RUNG wire#w3
   RUNG wire#w1
      Contact( #Dose.Dose_Stop.%X11 )
      wire#w4
      Coil( #Dose_Salt.ISTOP_AUT )
   END_RUNG
   RUNG wire#w1
      I_Contact( #State."Dose EN" )
      wire#w5
      Contact( #Dose_Salt.QHELD )
   END_RUNG wire#w4
   RUNG wire#w1
      I_Contact( #Dose.Dose_Prod_Ready.%X11 )
   END_RUNG wire#w5
   RUNG wire#w1
      Contact( #Dose_Salt.QDoseComplete )
      wire#w6
      Coil( #Dose_Salt.ICOMP_AUT )
   END_RUNG
   RUNG wire#w1
      Contact( #Dose_Salt.QSTOPPED )
   END_RUNG wire#w6
   // the same network as SCL:
   #Dose_Salt.ISTART_AUT := #AlwaysON AND #Dose.Dose_EN.%X4 AND #Dose.Dose_Tank_Available.%X11 AND (#Dose_Salt.SP_DOSEQTY > 0.0) AND #Dose.Dose_Start.%X11;
   IF #AlwaysON AND (NOT #Dose.Dose_EN.%X4 OR NOT #Dose.Dose_Tank_Available.%X11) THEN
       #Dose.Dose_Start.%X11 := FALSE;
   END_IF;
   #Dose_Salt.IHOLD_AUT := #AlwaysON AND (#Dose.Dose_Pause.%X11 OR NOT #State."Dose EN" OR NOT #Dose.Dose_Prod_Ready.%X11);
   #Dose_Salt.ISTOP_AUT := #AlwaysON AND (#Dose.Dose_Stop.%X11 OR ((NOT #State."Dose EN" OR NOT #Dose.Dose_Prod_Ready.%X11) AND #Dose_Salt.QHELD));
   #Dose_Salt.ICOMP_AUT := #AlwaysON AND (#Dose_Salt.QDoseComplete OR #Dose_Salt.QSTOPPED);
END_REGION

REGION Network 106: Dose Salt
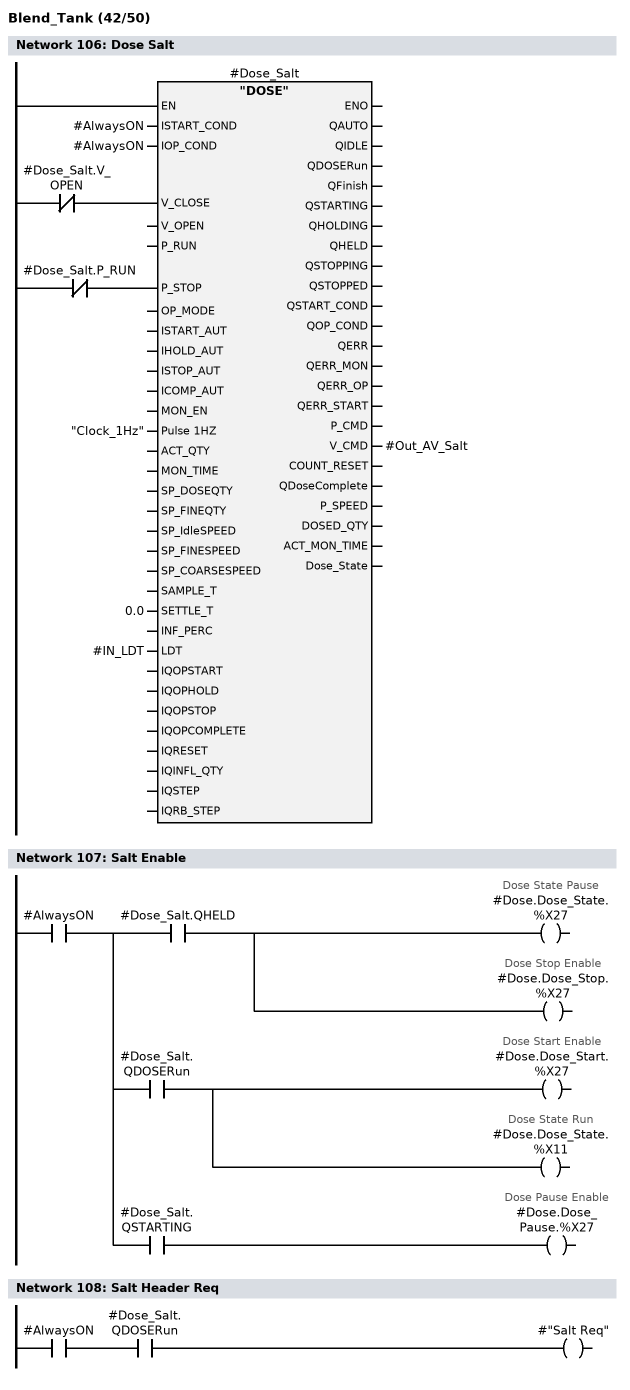
   RUNG wire#powerrail
      #Dose_Salt(V_CLOSE := wire#w1, P_STOP := wire#w2, ISTART_COND := #AlwaysON, IOP_COND := #AlwaysON, V_OPEN :=, P_RUN :=, OP_MODE :=, ISTART_AUT :=, IHOLD_AUT :=, ISTOP_AUT :=, ICOMP_AUT :=, MON_EN :=, "Pulse 1HZ" := "Clock_1Hz", ACT_QTY :=, MON_TIME :=, SP_DOSEQTY :=, SP_FINEQTY :=, SP_IdleSPEED :=, SP_FINESPEED :=, SP_COARSESPEED :=, SAMPLE_T :=, SETTLE_T := 0.0, INF_PERC :=, LDT := #IN_LDT, IQOPSTART :=, IQOPHOLD :=, IQOPSTOP :=, IQOPCOMPLETE :=, IQRESET :=, IQINFL_QTY :=, IQSTEP :=, IQRB_STEP :=, QAUTO =>, QIDLE =>, QDOSERun =>, QFinish =>, QSTARTING =>, QHOLDING =>, QHELD =>, QSTOPPING =>, QSTOPPED =>, QSTART_COND =>, QOP_COND =>, QERR =>, QERR_MON =>, QERR_OP =>, QERR_START =>, P_CMD =>, V_CMD => #Out_AV_Salt, COUNT_RESET =>, QDoseComplete =>, P_SPEED =>, DOSED_QTY =>, ACT_MON_TIME =>, Dose_State =>)
   END_RUNG
   RUNG wire#powerrail
      I_Contact( #Dose_Salt.V_OPEN )
   END_RUNG wire#w1
   RUNG wire#powerrail
      I_Contact( #Dose_Salt.P_RUN )
   END_RUNG wire#w2
   // the same network as SCL:
   #Dose_Salt(ISTART_COND := #AlwaysON,   // "DOSE"
              IOP_COND := #AlwaysON,
              V_CLOSE := NOT #Dose_Salt.V_OPEN,
              P_STOP := NOT #Dose_Salt.P_RUN,
              "Pulse 1HZ" := "Clock_1Hz",
              SETTLE_T := 0.0,
              LDT := #IN_LDT,
              V_CMD => #Out_AV_Salt);
END_REGION

REGION Network 107: Salt Enable
   RUNG wire#powerrail
      Contact( #AlwaysON )
      wire#w1
      Contact( #Dose_Salt.QHELD )
      wire#w2
      Coil( #Dose.Dose_State.%X27 )   // Dose State Pause
   END_RUNG
   RUNG wire#w2
      Coil( #Dose.Dose_Stop.%X27 )   // Dose Stop Enable
   END_RUNG
   RUNG wire#w1
      Contact( #Dose_Salt.QDOSERun )
      wire#w3
      Coil( #Dose.Dose_Start.%X27 )   // Dose Start Enable
   END_RUNG
   RUNG wire#w3
      Coil( #Dose.Dose_State.%X11 )   // Dose State Run
   END_RUNG
   RUNG wire#w1
      Contact( #Dose_Salt.QSTARTING )
      Coil( #Dose.Dose_Pause.%X27 )   // Dose Pause Enable
   END_RUNG
   // the same network as SCL:
   #Dose.Dose_State.%X27 := #AlwaysON AND #Dose_Salt.QHELD;   // Dose State Pause
   #Dose.Dose_Stop.%X27 := #Dose.Dose_State.%X27;   // Dose Stop Enable
   #Dose.Dose_Start.%X27 := #AlwaysON AND #Dose_Salt.QDOSERun;   // Dose Start Enable
   #Dose.Dose_State.%X11 := #Dose.Dose_Start.%X27;   // Dose State Run
   #Dose.Dose_Pause.%X27 := #AlwaysON AND #Dose_Salt.QSTARTING;   // Dose Pause Enable
END_REGION

REGION Network 108: Salt Header Req
   RUNG wire#powerrail
      Contact( #AlwaysON )
      Contact( #Dose_Salt.QDOSERun )
      Coil( #"Salt Req" )
   END_RUNG
   // the same network as SCL:
   #"Salt Req" := #AlwaysON AND #Dose_Salt.QDOSERun;
END_REGION

REGION Network 110: ProWater Setpoint
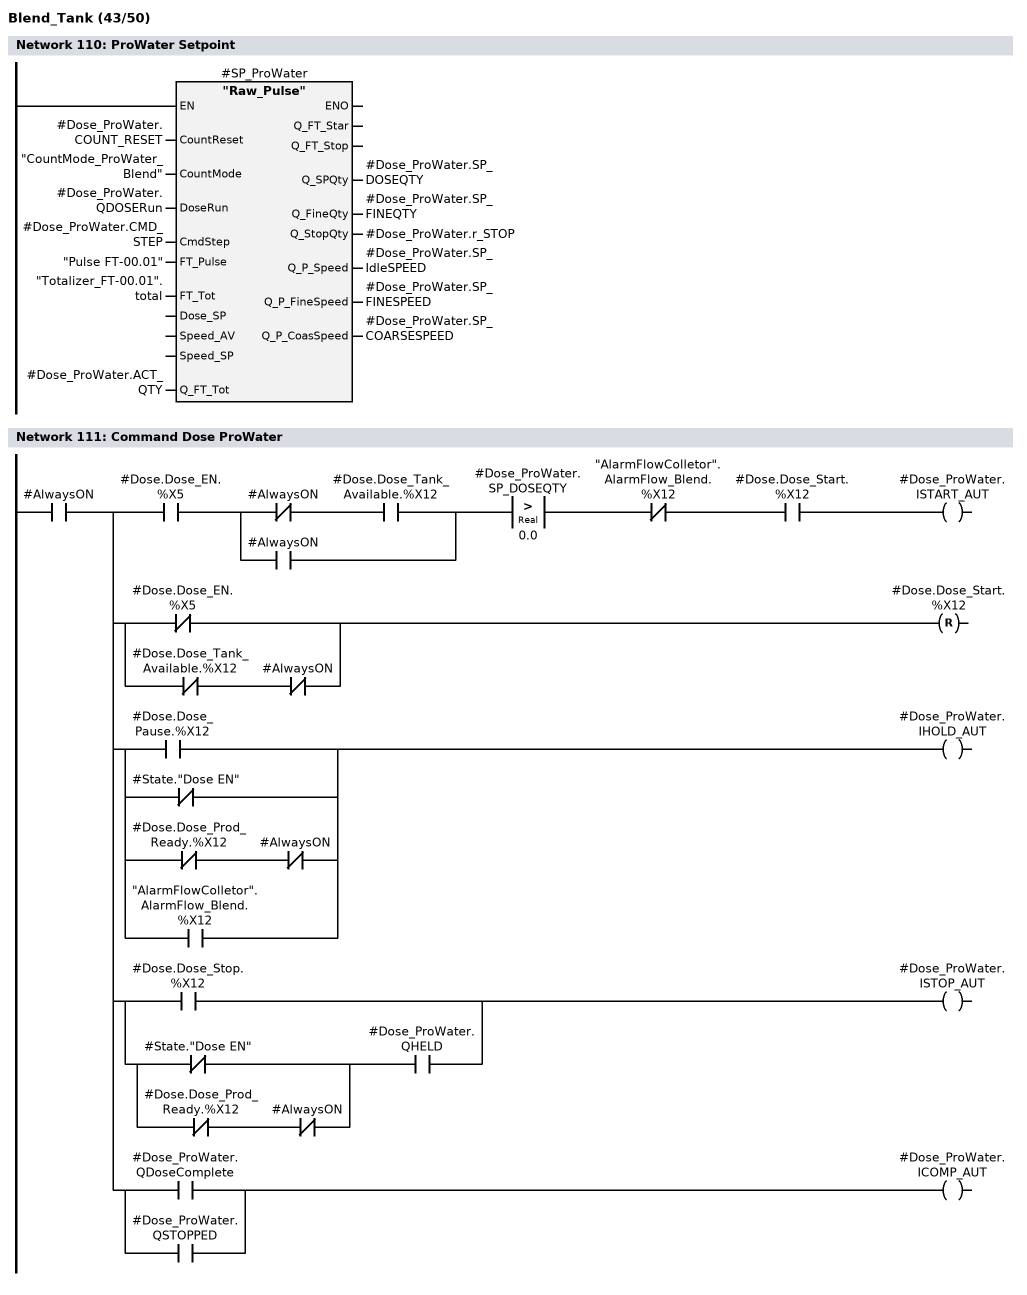
   RUNG wire#powerrail
      #SP_ProWater(CountReset := #Dose_ProWater.COUNT_RESET, CountMode := "CountMode_ProWater_Blend", DoseRun := #Dose_ProWater.QDOSERun, CmdStep := #Dose_ProWater.CMD_STEP, FT_Pulse := "Pulse FT-00.01", FT_Tot := "Totalizer_FT-00.01".total, Dose_SP :=, Speed_AV :=, Speed_SP :=, Q_FT_Tot := #Dose_ProWater.ACT_QTY, Q_FT_Star =>, Q_FT_Stop =>, Q_SPQty => #Dose_ProWater.SP_DOSEQTY, Q_FineQty => #Dose_ProWater.SP_FINEQTY, Q_StopQty => #Dose_ProWater.r_STOP, Q_P_Speed => #Dose_ProWater.SP_IdleSPEED, Q_P_FineSpeed => #Dose_ProWater.SP_FINESPEED, Q_P_CoasSpeed => #Dose_ProWater.SP_COARSESPEED)
   END_RUNG
   // the same network as SCL:
   #SP_ProWater(CountReset := #Dose_ProWater.COUNT_RESET,   // "Raw_Pulse"
                CountMode := "CountMode_ProWater_Blend",
                DoseRun := #Dose_ProWater.QDOSERun,
                CmdStep := #Dose_ProWater.CMD_STEP,
                FT_Pulse := "Pulse FT-00.01",
                FT_Tot := "Totalizer_FT-00.01".total,
                Q_FT_Tot := #Dose_ProWater.ACT_QTY,
                Q_SPQty => #Dose_ProWater.SP_DOSEQTY,
                Q_FineQty => #Dose_ProWater.SP_FINEQTY,
                Q_StopQty => #Dose_ProWater.r_STOP,
                Q_P_Speed => #Dose_ProWater.SP_IdleSPEED,
                Q_P_FineSpeed => #Dose_ProWater.SP_FINESPEED,
                Q_P_CoasSpeed => #Dose_ProWater.SP_COARSESPEED);
END_REGION

REGION Network 111: Command Dose ProWater
   RUNG wire#powerrail
      Contact( #AlwaysON )
      wire#w1
      Contact( #Dose.Dose_EN.%X5 )
      wire#w2
      I_Contact( #AlwaysON )
      Contact( #Dose.Dose_Tank_Available.%X12 )
      wire#w3
      { S7_Templates := "SrcType := Real" } GT_Contact(in1 := #Dose_ProWater.SP_DOSEQTY, in2 := 0.0)
      I_Contact( "AlarmFlowColletor".AlarmFlow_Blend.%X12 )
      Contact( #Dose.Dose_Start.%X12 )
      Coil( #Dose_ProWater.ISTART_AUT )
   END_RUNG
   RUNG wire#w2
      Contact( #AlwaysON )
   END_RUNG wire#w3
   RUNG wire#w1
      I_Contact( #Dose.Dose_EN.%X5 )
      wire#w4
      R_Coil( #Dose.Dose_Start.%X12 )
   END_RUNG
   RUNG wire#w1
      I_Contact( #Dose.Dose_Tank_Available.%X12 )
      I_Contact( #AlwaysON )
   END_RUNG wire#w4
   RUNG wire#w1
      Contact( #Dose.Dose_Pause.%X12 )
      wire#w5
      Coil( #Dose_ProWater.IHOLD_AUT )
   END_RUNG
   RUNG wire#w1
      I_Contact( #State."Dose EN" )
   END_RUNG wire#w5
   RUNG wire#w1
      I_Contact( #Dose.Dose_Prod_Ready.%X12 )
      I_Contact( #AlwaysON )
   END_RUNG wire#w5
   RUNG wire#w1
      Contact( "AlarmFlowColletor".AlarmFlow_Blend.%X12 )
   END_RUNG wire#w5
   RUNG wire#w1
      Contact( #Dose.Dose_Stop.%X12 )
      wire#w6
      Coil( #Dose_ProWater.ISTOP_AUT )
   END_RUNG
   RUNG wire#w1
      I_Contact( #State."Dose EN" )
      wire#w7
      Contact( #Dose_ProWater.QHELD )
   END_RUNG wire#w6
   RUNG wire#w1
      I_Contact( #Dose.Dose_Prod_Ready.%X12 )
      I_Contact( #AlwaysON )
   END_RUNG wire#w7
   RUNG wire#w1
      Contact( #Dose_ProWater.QDoseComplete )
      wire#w8
      Coil( #Dose_ProWater.ICOMP_AUT )
   END_RUNG
   RUNG wire#w1
      Contact( #Dose_ProWater.QSTOPPED )
   END_RUNG wire#w8
   // the same network as SCL:
   #Dose_ProWater.ISTART_AUT := #AlwaysON AND #Dose.Dose_EN.%X5 AND ((NOT #AlwaysON AND #Dose.Dose_Tank_Available.%X12) OR #AlwaysON) AND (#Dose_ProWater.SP_DOSEQTY > 0.0) AND NOT "AlarmFlowColletor".AlarmFlow_Blend.%X12 AND #Dose.Dose_Start.%X12;
   IF #AlwaysON AND (NOT #Dose.Dose_EN.%X5 OR (NOT #Dose.Dose_Tank_Available.%X12 AND NOT #AlwaysON)) THEN
       #Dose.Dose_Start.%X12 := FALSE;
   END_IF;
   #Dose_ProWater.IHOLD_AUT := #AlwaysON AND (#Dose.Dose_Pause.%X12 OR NOT #State."Dose EN" OR (NOT #Dose.Dose_Prod_Ready.%X12 AND NOT #AlwaysON) OR "AlarmFlowColletor".AlarmFlow_Blend.%X12);
   #Dose_ProWater.ISTOP_AUT := #AlwaysON AND (#Dose.Dose_Stop.%X12 OR ((NOT #State."Dose EN" OR (NOT #Dose.Dose_Prod_Ready.%X12 AND NOT #AlwaysON)) AND #Dose_ProWater.QHELD));
   #Dose_ProWater.ICOMP_AUT := #AlwaysON AND (#Dose_ProWater.QDoseComplete OR #Dose_ProWater.QSTOPPED);
END_REGION

REGION Network 112: Dose ProWater
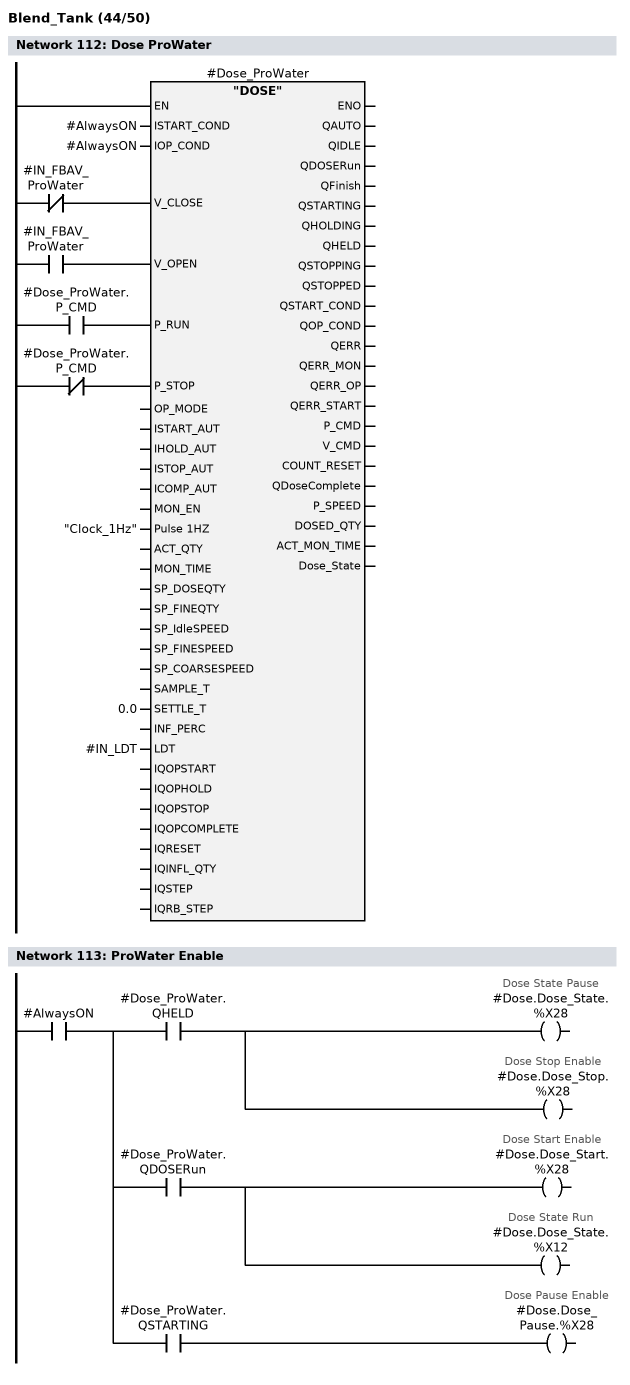
   RUNG wire#powerrail
      #Dose_ProWater(V_CLOSE := wire#w1, V_OPEN := wire#w2, P_RUN := wire#w3, P_STOP := wire#w4, ISTART_COND := #AlwaysON, IOP_COND := #AlwaysON, OP_MODE :=, ISTART_AUT :=, IHOLD_AUT :=, ISTOP_AUT :=, ICOMP_AUT :=, MON_EN :=, "Pulse 1HZ" := "Clock_1Hz", ACT_QTY :=, MON_TIME :=, SP_DOSEQTY :=, SP_FINEQTY :=, SP_IdleSPEED :=, SP_FINESPEED :=, SP_COARSESPEED :=, SAMPLE_T :=, SETTLE_T := 0.0, INF_PERC :=, LDT := #IN_LDT, IQOPSTART :=, IQOPHOLD :=, IQOPSTOP :=, IQOPCOMPLETE :=, IQRESET :=, IQINFL_QTY :=, IQSTEP :=, IQRB_STEP :=, QAUTO =>, QIDLE =>, QDOSERun =>, QFinish =>, QSTARTING =>, QHOLDING =>, QHELD =>, QSTOPPING =>, QSTOPPED =>, QSTART_COND =>, QOP_COND =>, QERR =>, QERR_MON =>, QERR_OP =>, QERR_START =>, P_CMD =>, V_CMD =>, COUNT_RESET =>, QDoseComplete =>, P_SPEED =>, DOSED_QTY =>, ACT_MON_TIME =>, Dose_State =>)
   END_RUNG
   RUNG wire#powerrail
      I_Contact( #IN_FBAV_ProWater )
   END_RUNG wire#w1
   RUNG wire#powerrail
      Contact( #IN_FBAV_ProWater )
   END_RUNG wire#w2
   RUNG wire#powerrail
      Contact( #Dose_ProWater.P_CMD )
   END_RUNG wire#w3
   RUNG wire#powerrail
      I_Contact( #Dose_ProWater.P_CMD )
   END_RUNG wire#w4
   // the same network as SCL:
   #Dose_ProWater(ISTART_COND := #AlwaysON,   // "DOSE"
                  IOP_COND := #AlwaysON,
                  V_CLOSE := NOT #IN_FBAV_ProWater,
                  V_OPEN := #IN_FBAV_ProWater,
                  P_RUN := #Dose_ProWater.P_CMD,
                  P_STOP := NOT #Dose_ProWater.P_CMD,
                  "Pulse 1HZ" := "Clock_1Hz",
                  SETTLE_T := 0.0,
                  LDT := #IN_LDT);
END_REGION

REGION Network 113: ProWater Enable
   RUNG wire#powerrail
      Contact( #AlwaysON )
      wire#w1
      Contact( #Dose_ProWater.QHELD )
      wire#w2
      Coil( #Dose.Dose_State.%X28 )   // Dose State Pause
   END_RUNG
   RUNG wire#w2
      Coil( #Dose.Dose_Stop.%X28 )   // Dose Stop Enable
   END_RUNG
   RUNG wire#w1
      Contact( #Dose_ProWater.QDOSERun )
      wire#w3
      Coil( #Dose.Dose_Start.%X28 )   // Dose Start Enable
   END_RUNG
   RUNG wire#w3
      Coil( #Dose.Dose_State.%X12 )   // Dose State Run
   END_RUNG
   RUNG wire#w1
      Contact( #Dose_ProWater.QSTARTING )
      Coil( #Dose.Dose_Pause.%X28 )   // Dose Pause Enable
   END_RUNG
   // the same network as SCL:
   #Dose.Dose_State.%X28 := #AlwaysON AND #Dose_ProWater.QHELD;   // Dose State Pause
   #Dose.Dose_Stop.%X28 := #Dose.Dose_State.%X28;   // Dose Stop Enable
   #Dose.Dose_Start.%X28 := #AlwaysON AND #Dose_ProWater.QDOSERun;   // Dose Start Enable
   #Dose.Dose_State.%X12 := #Dose.Dose_Start.%X28;   // Dose State Run
   #Dose.Dose_Pause.%X28 := #AlwaysON AND #Dose_ProWater.QSTARTING;   // Dose Pause Enable
END_REGION

REGION Network 114: ProWater Header Req & Valve
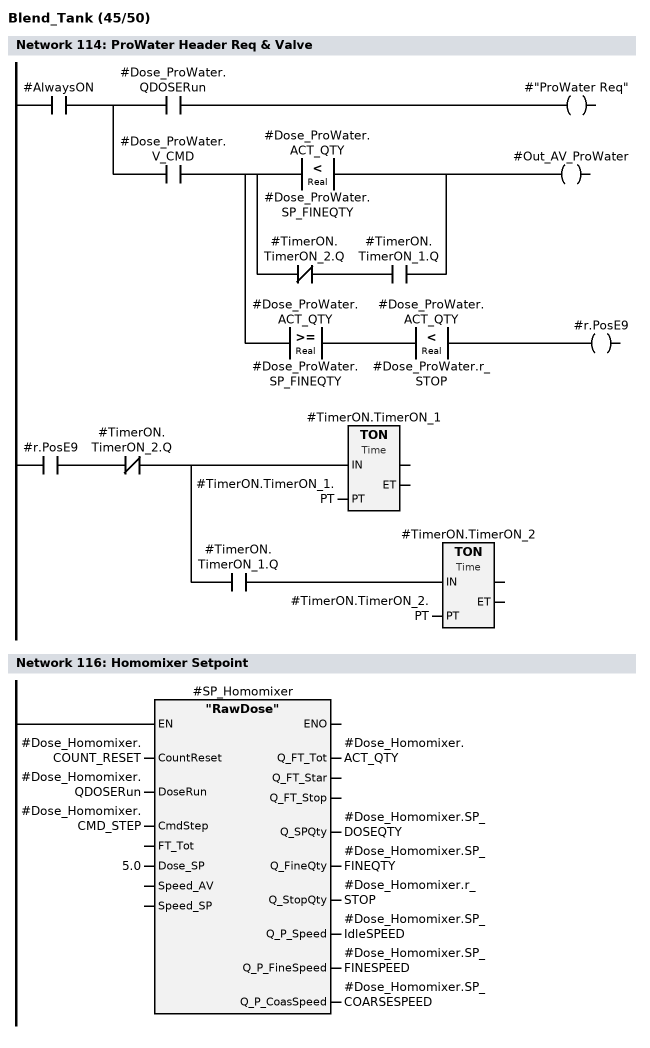
   RUNG wire#powerrail
      Contact( #AlwaysON )
      wire#w1
      Contact( #Dose_ProWater.QDOSERun )
      Coil( #"ProWater Req" )
   END_RUNG
   RUNG wire#w1
      Contact( #Dose_ProWater.V_CMD )
      wire#w2
      { S7_Templates := "SrcType := Real" } LT_Contact(in1 := #Dose_ProWater.ACT_QTY, in2 := #Dose_ProWater.SP_FINEQTY)
      wire#w3
      Coil( #Out_AV_ProWater )
   END_RUNG
   RUNG wire#w2
      I_Contact( #TimerON.TimerON_2.Q )
      Contact( #TimerON.TimerON_1.Q )
   END_RUNG wire#w3
   RUNG wire#w2
      { S7_Templates := "SrcType := Real" } GE_Contact(in1 := #Dose_ProWater.ACT_QTY, in2 := #Dose_ProWater.SP_FINEQTY)
      { S7_Templates := "SrcType := Real" } LT_Contact(in1 := #Dose_ProWater.ACT_QTY, in2 := #Dose_ProWater.r_STOP)
      Coil( #r.PosE9 )
   END_RUNG
   RUNG wire#powerrail
      Contact( #r.PosE9 )
      I_Contact( #TimerON.TimerON_2.Q )
      wire#w4
      { S7_Templates := "time_type := Time" } #TimerON.TimerON_1.TON(pt := #TimerON.TimerON_1.PT, et =>)
   END_RUNG
   RUNG wire#w4
      Contact( #TimerON.TimerON_1.Q )
      { S7_Templates := "time_type := Time" } #TimerON.TimerON_2.TON(pt := #TimerON.TimerON_2.PT, et =>)
   END_RUNG
   // the same network as SCL:
   #"ProWater Req" := #AlwaysON AND #Dose_ProWater.QDOSERun;
   #_w1 := #AlwaysON AND #Dose_ProWater.V_CMD;
   #Out_AV_ProWater := #_w1 AND ((#Dose_ProWater.ACT_QTY < #Dose_ProWater.SP_FINEQTY) OR (NOT #TimerON.TimerON_2.Q AND #TimerON.TimerON_1.Q));
   #r.PosE9 := #_w1 AND (#Dose_ProWater.ACT_QTY >= #Dose_ProWater.SP_FINEQTY) AND (#Dose_ProWater.ACT_QTY < #Dose_ProWater.r_STOP);
   #_w2 := #r.PosE9 AND NOT #TimerON.TimerON_2.Q;
   #TimerON.TimerON_1.TON(IN := #_w2, PT := #TimerON.TimerON_1.PT);
   #TimerON.TimerON_2.TON(IN := #_w2 AND #TimerON.TimerON_1.Q, PT := #TimerON.TimerON_2.PT);
END_REGION

REGION Network 116: Homomixer Setpoint
   RUNG wire#powerrail
      #SP_Homomixer(CountReset := #Dose_Homomixer.COUNT_RESET, DoseRun := #Dose_Homomixer.QDOSERun, CmdStep := #Dose_Homomixer.CMD_STEP, FT_Tot :=, Dose_SP := 5.0, Speed_AV :=, Speed_SP :=, Q_FT_Tot => #Dose_Homomixer.ACT_QTY, Q_FT_Star =>, Q_FT_Stop =>, Q_SPQty => #Dose_Homomixer.SP_DOSEQTY, Q_FineQty => #Dose_Homomixer.SP_FINEQTY, Q_StopQty => #Dose_Homomixer.r_STOP, Q_P_Speed => #Dose_Homomixer.SP_IdleSPEED, Q_P_FineSpeed => #Dose_Homomixer.SP_FINESPEED, Q_P_CoasSpeed => #Dose_Homomixer.SP_COARSESPEED)
   END_RUNG
   // the same network as SCL:
   #SP_Homomixer(CountReset := #Dose_Homomixer.COUNT_RESET,   // "RawDose"
                 DoseRun := #Dose_Homomixer.QDOSERun,
                 CmdStep := #Dose_Homomixer.CMD_STEP,
                 Dose_SP := 5.0,
                 Q_FT_Tot => #Dose_Homomixer.ACT_QTY,
                 Q_SPQty => #Dose_Homomixer.SP_DOSEQTY,
                 Q_FineQty => #Dose_Homomixer.SP_FINEQTY,
                 Q_StopQty => #Dose_Homomixer.r_STOP,
                 Q_P_Speed => #Dose_Homomixer.SP_IdleSPEED,
                 Q_P_FineSpeed => #Dose_Homomixer.SP_FINESPEED,
                 Q_P_CoasSpeed => #Dose_Homomixer.SP_COARSESPEED);
END_REGION

REGION Network 117: Command Dose Homomixer
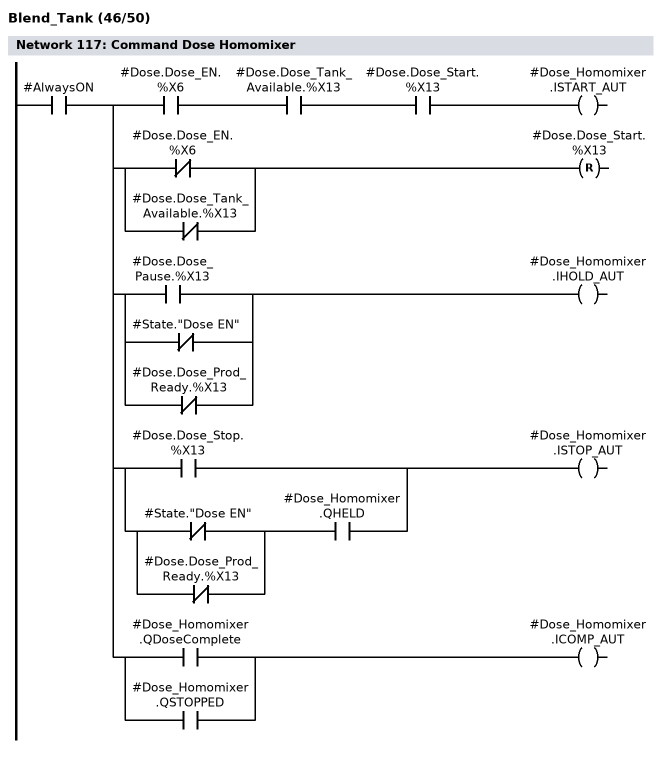
   RUNG wire#powerrail
      Contact( #AlwaysON )
      wire#w1
      Contact( #Dose.Dose_EN.%X6 )
      Contact( #Dose.Dose_Tank_Available.%X13 )
      Contact( #Dose.Dose_Start.%X13 )
      Coil( #Dose_Homomixer.ISTART_AUT )
   END_RUNG
   RUNG wire#w1
      I_Contact( #Dose.Dose_EN.%X6 )
      wire#w2
      R_Coil( #Dose.Dose_Start.%X13 )
   END_RUNG
   RUNG wire#w1
      I_Contact( #Dose.Dose_Tank_Available.%X13 )
   END_RUNG wire#w2
   RUNG wire#w1
      Contact( #Dose.Dose_Pause.%X13 )
      wire#w3
      Coil( #Dose_Homomixer.IHOLD_AUT )
   END_RUNG
   RUNG wire#w1
      I_Contact( #State."Dose EN" )
   END_RUNG wire#w3
   RUNG wire#w1
      I_Contact( #Dose.Dose_Prod_Ready.%X13 )
   END_RUNG wire#w3
   RUNG wire#w1
      Contact( #Dose.Dose_Stop.%X13 )
      wire#w4
      Coil( #Dose_Homomixer.ISTOP_AUT )
   END_RUNG
   RUNG wire#w1
      I_Contact( #State."Dose EN" )
      wire#w5
      Contact( #Dose_Homomixer.QHELD )
   END_RUNG wire#w4
   RUNG wire#w1
      I_Contact( #Dose.Dose_Prod_Ready.%X13 )
   END_RUNG wire#w5
   RUNG wire#w1
      Contact( #Dose_Homomixer.QDoseComplete )
      wire#w6
      Coil( #Dose_Homomixer.ICOMP_AUT )
   END_RUNG
   RUNG wire#w1
      Contact( #Dose_Homomixer.QSTOPPED )
   END_RUNG wire#w6
   // the same network as SCL:
   #Dose_Homomixer.ISTART_AUT := #AlwaysON AND #Dose.Dose_EN.%X6 AND #Dose.Dose_Tank_Available.%X13 AND #Dose.Dose_Start.%X13;
   IF #AlwaysON AND (NOT #Dose.Dose_EN.%X6 OR NOT #Dose.Dose_Tank_Available.%X13) THEN
       #Dose.Dose_Start.%X13 := FALSE;
   END_IF;
   #Dose_Homomixer.IHOLD_AUT := #AlwaysON AND (#Dose.Dose_Pause.%X13 OR NOT #State."Dose EN" OR NOT #Dose.Dose_Prod_Ready.%X13);
   #Dose_Homomixer.ISTOP_AUT := #AlwaysON AND (#Dose.Dose_Stop.%X13 OR ((NOT #State."Dose EN" OR NOT #Dose.Dose_Prod_Ready.%X13) AND #Dose_Homomixer.QHELD));
   #Dose_Homomixer.ICOMP_AUT := #AlwaysON AND (#Dose_Homomixer.QDoseComplete OR #Dose_Homomixer.QSTOPPED);
END_REGION

REGION Network 118: Dose Homomixer
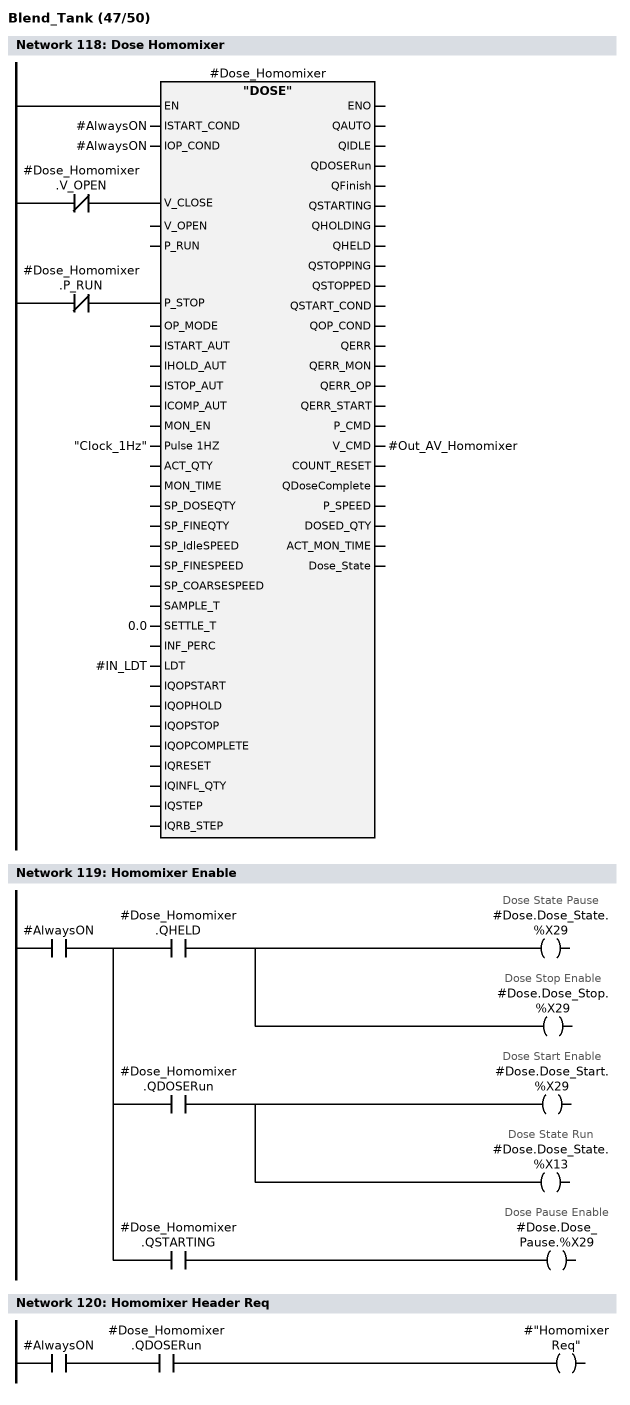
   RUNG wire#powerrail
      #Dose_Homomixer(V_CLOSE := wire#w1, P_STOP := wire#w2, ISTART_COND := #AlwaysON, IOP_COND := #AlwaysON, V_OPEN :=, P_RUN :=, OP_MODE :=, ISTART_AUT :=, IHOLD_AUT :=, ISTOP_AUT :=, ICOMP_AUT :=, MON_EN :=, "Pulse 1HZ" := "Clock_1Hz", ACT_QTY :=, MON_TIME :=, SP_DOSEQTY :=, SP_FINEQTY :=, SP_IdleSPEED :=, SP_FINESPEED :=, SP_COARSESPEED :=, SAMPLE_T :=, SETTLE_T := 0.0, INF_PERC :=, LDT := #IN_LDT, IQOPSTART :=, IQOPHOLD :=, IQOPSTOP :=, IQOPCOMPLETE :=, IQRESET :=, IQINFL_QTY :=, IQSTEP :=, IQRB_STEP :=, QAUTO =>, QIDLE =>, QDOSERun =>, QFinish =>, QSTARTING =>, QHOLDING =>, QHELD =>, QSTOPPING =>, QSTOPPED =>, QSTART_COND =>, QOP_COND =>, QERR =>, QERR_MON =>, QERR_OP =>, QERR_START =>, P_CMD =>, V_CMD => #Out_AV_Homomixer, COUNT_RESET =>, QDoseComplete =>, P_SPEED =>, DOSED_QTY =>, ACT_MON_TIME =>, Dose_State =>)
   END_RUNG
   RUNG wire#powerrail
      I_Contact( #Dose_Homomixer.V_OPEN )
   END_RUNG wire#w1
   RUNG wire#powerrail
      I_Contact( #Dose_Homomixer.P_RUN )
   END_RUNG wire#w2
   // the same network as SCL:
   #Dose_Homomixer(ISTART_COND := #AlwaysON,   // "DOSE"
                   IOP_COND := #AlwaysON,
                   V_CLOSE := NOT #Dose_Homomixer.V_OPEN,
                   P_STOP := NOT #Dose_Homomixer.P_RUN,
                   "Pulse 1HZ" := "Clock_1Hz",
                   SETTLE_T := 0.0,
                   LDT := #IN_LDT,
                   V_CMD => #Out_AV_Homomixer);
END_REGION

REGION Network 119: Homomixer Enable
   RUNG wire#powerrail
      Contact( #AlwaysON )
      wire#w1
      Contact( #Dose_Homomixer.QHELD )
      wire#w2
      Coil( #Dose.Dose_State.%X29 )   // Dose State Pause
   END_RUNG
   RUNG wire#w2
      Coil( #Dose.Dose_Stop.%X29 )   // Dose Stop Enable
   END_RUNG
   RUNG wire#w1
      Contact( #Dose_Homomixer.QDOSERun )
      wire#w3
      Coil( #Dose.Dose_Start.%X29 )   // Dose Start Enable
   END_RUNG
   RUNG wire#w3
      Coil( #Dose.Dose_State.%X13 )   // Dose State Run
   END_RUNG
   RUNG wire#w1
      Contact( #Dose_Homomixer.QSTARTING )
      Coil( #Dose.Dose_Pause.%X29 )   // Dose Pause Enable
   END_RUNG
   // the same network as SCL:
   #Dose.Dose_State.%X29 := #AlwaysON AND #Dose_Homomixer.QHELD;   // Dose State Pause
   #Dose.Dose_Stop.%X29 := #Dose.Dose_State.%X29;   // Dose Stop Enable
   #Dose.Dose_Start.%X29 := #AlwaysON AND #Dose_Homomixer.QDOSERun;   // Dose Start Enable
   #Dose.Dose_State.%X13 := #Dose.Dose_Start.%X29;   // Dose State Run
   #Dose.Dose_Pause.%X29 := #AlwaysON AND #Dose_Homomixer.QSTARTING;   // Dose Pause Enable
END_REGION

REGION Network 120: Homomixer Header Req
   RUNG wire#powerrail
      Contact( #AlwaysON )
      Contact( #Dose_Homomixer.QDOSERun )
      Coil( #"Homomixer Req" )
   END_RUNG
   // the same network as SCL:
   #"Homomixer Req" := #AlwaysON AND #Dose_Homomixer.QDOSERun;
END_REGION

REGION Network 122: Level Scaling
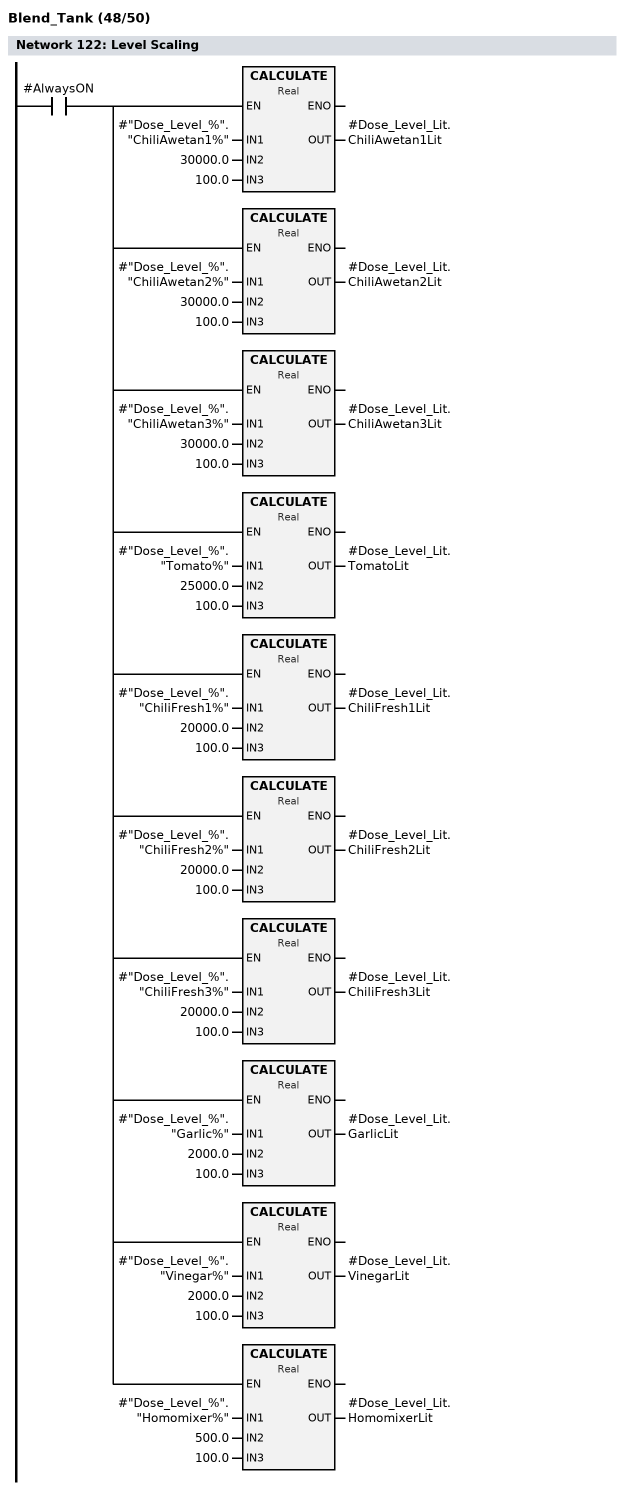
   RUNG wire#powerrail
      Contact( #AlwaysON )
      wire#w1
      { S7_Templates := "SrcType := Real"; S7_Expression := "(IN1 * IN2) / IN3" } Calculate(in1 := #"Dose_Level_%"."ChiliAwetan1%", in2 := 30000.0, in3 := 100.0, out => #Dose_Level_Lit.ChiliAwetan1Lit)
   END_RUNG
   RUNG wire#w1
      { S7_Templates := "SrcType := Real"; S7_Expression := "(IN1 * IN2) / IN3" } Calculate(in1 := #"Dose_Level_%"."ChiliAwetan2%", in2 := 30000.0, in3 := 100.0, out => #Dose_Level_Lit.ChiliAwetan2Lit)
   END_RUNG
   RUNG wire#w1
      { S7_Templates := "SrcType := Real"; S7_Expression := "(IN1 * IN2) / IN3" } Calculate(in1 := #"Dose_Level_%"."ChiliAwetan3%", in2 := 30000.0, in3 := 100.0, out => #Dose_Level_Lit.ChiliAwetan3Lit)
   END_RUNG
   RUNG wire#w1
      { S7_Templates := "SrcType := Real"; S7_Expression := "(IN1 * IN2) / IN3" } Calculate(in1 := #"Dose_Level_%"."Tomato%", in2 := 25000.0, in3 := 100.0, out => #Dose_Level_Lit.TomatoLit)
   END_RUNG
   RUNG wire#w1
      { S7_Templates := "SrcType := Real"; S7_Expression := "(IN1 * IN2) / IN3" } Calculate(in1 := #"Dose_Level_%"."ChiliFresh1%", in2 := 20000.0, in3 := 100.0, out => #Dose_Level_Lit.ChiliFresh1Lit)
   END_RUNG
   RUNG wire#w1
      { S7_Templates := "SrcType := Real"; S7_Expression := "(IN1 * IN2) / IN3" } Calculate(in1 := #"Dose_Level_%"."ChiliFresh2%", in2 := 20000.0, in3 := 100.0, out => #Dose_Level_Lit.ChiliFresh2Lit)
   END_RUNG
   RUNG wire#w1
      { S7_Templates := "SrcType := Real"; S7_Expression := "(IN1 * IN2) / IN3" } Calculate(in1 := #"Dose_Level_%"."ChiliFresh3%", in2 := 20000.0, in3 := 100.0, out => #Dose_Level_Lit.ChiliFresh3Lit)
   END_RUNG
   RUNG wire#w1
      { S7_Templates := "SrcType := Real"; S7_Expression := "(IN1 * IN2) / IN3" } Calculate(in1 := #"Dose_Level_%"."Garlic%", in2 := 2000.0, in3 := 100.0, out => #Dose_Level_Lit.GarlicLit)
   END_RUNG
   RUNG wire#w1
      { S7_Templates := "SrcType := Real"; S7_Expression := "(IN1 * IN2) / IN3" } Calculate(in1 := #"Dose_Level_%"."Vinegar%", in2 := 2000.0, in3 := 100.0, out => #Dose_Level_Lit.VinegarLit)
   END_RUNG
   RUNG wire#w1
      { S7_Templates := "SrcType := Real"; S7_Expression := "(IN1 * IN2) / IN3" } Calculate(in1 := #"Dose_Level_%"."Homomixer%", in2 := 500.0, in3 := 100.0, out => #Dose_Level_Lit.HomomixerLit)
   END_RUNG
   // the same network as SCL:
   IF #AlwaysON THEN
       #Dose_Level_Lit.ChiliAwetan1Lit := (#"Dose_Level_%"."ChiliAwetan1%" * 30000.0) / 100.0;
       #Dose_Level_Lit.ChiliAwetan2Lit := (#"Dose_Level_%"."ChiliAwetan2%" * 30000.0) / 100.0;
       #Dose_Level_Lit.ChiliAwetan3Lit := (#"Dose_Level_%"."ChiliAwetan3%" * 30000.0) / 100.0;
       #Dose_Level_Lit.TomatoLit := (#"Dose_Level_%"."Tomato%" * 25000.0) / 100.0;
       #Dose_Level_Lit.ChiliFresh1Lit := (#"Dose_Level_%"."ChiliFresh1%" * 20000.0) / 100.0;
       #Dose_Level_Lit.ChiliFresh2Lit := (#"Dose_Level_%"."ChiliFresh2%" * 20000.0) / 100.0;
       #Dose_Level_Lit.ChiliFresh3Lit := (#"Dose_Level_%"."ChiliFresh3%" * 20000.0) / 100.0;
       #Dose_Level_Lit.GarlicLit := (#"Dose_Level_%"."Garlic%" * 2000.0) / 100.0;
       #Dose_Level_Lit.VinegarLit := (#"Dose_Level_%"."Vinegar%" * 2000.0) / 100.0;
       #Dose_Level_Lit.HomomixerLit := (#"Dose_Level_%"."Homomixer%" * 500.0) / 100.0;
   END_IF;
END_REGION

REGION Network 123: Last Dose Qty
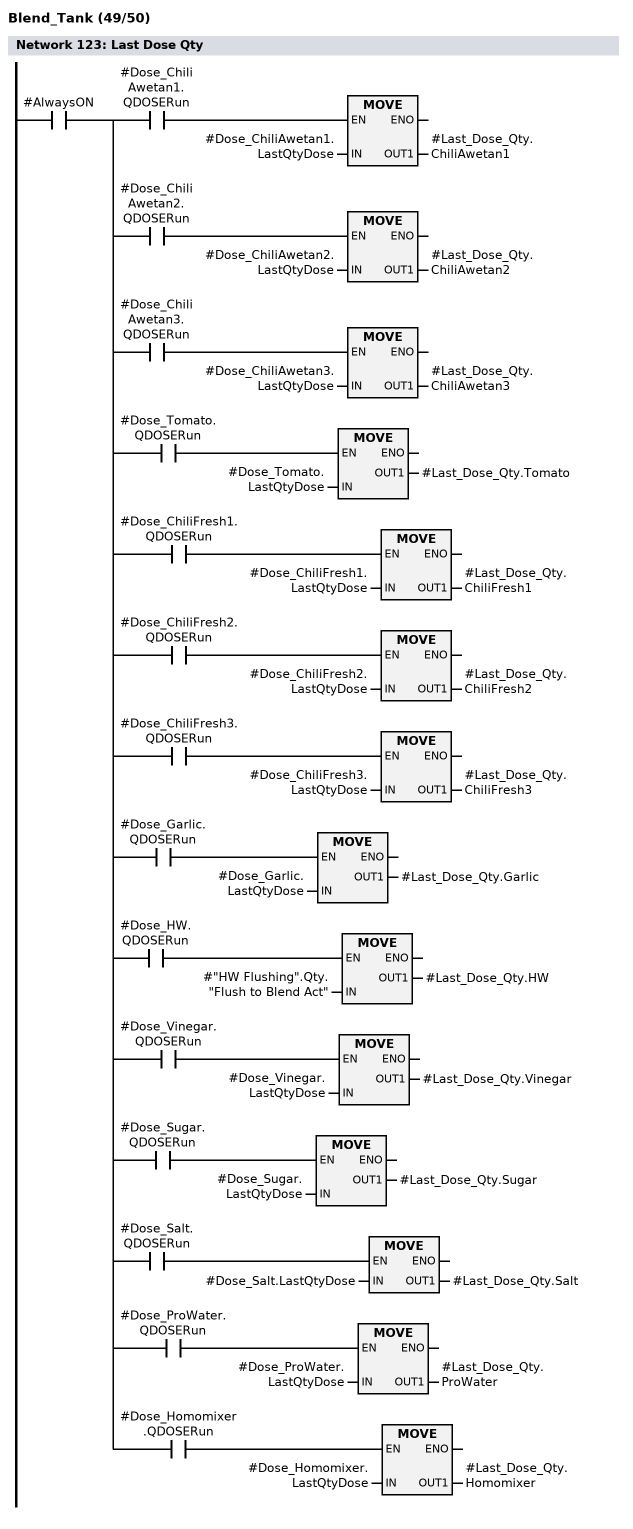
   RUNG wire#powerrail
      Contact( #AlwaysON )
      wire#w1
      Contact( #Dose_ChiliAwetan1.QDOSERun )
      Move(in := #Dose_ChiliAwetan1.LastQtyDose, out1 => #Last_Dose_Qty.ChiliAwetan1)
   END_RUNG
   RUNG wire#w1
      Contact( #Dose_ChiliAwetan2.QDOSERun )
      Move(in := #Dose_ChiliAwetan2.LastQtyDose, out1 => #Last_Dose_Qty.ChiliAwetan2)
   END_RUNG
   RUNG wire#w1
      Contact( #Dose_ChiliAwetan3.QDOSERun )
      Move(in := #Dose_ChiliAwetan3.LastQtyDose, out1 => #Last_Dose_Qty.ChiliAwetan3)
   END_RUNG
   RUNG wire#w1
      Contact( #Dose_Tomato.QDOSERun )
      Move(in := #Dose_Tomato.LastQtyDose, out1 => #Last_Dose_Qty.Tomato)
   END_RUNG
   RUNG wire#w1
      Contact( #Dose_ChiliFresh1.QDOSERun )
      Move(in := #Dose_ChiliFresh1.LastQtyDose, out1 => #Last_Dose_Qty.ChiliFresh1)
   END_RUNG
   RUNG wire#w1
      Contact( #Dose_ChiliFresh2.QDOSERun )
      Move(in := #Dose_ChiliFresh2.LastQtyDose, out1 => #Last_Dose_Qty.ChiliFresh2)
   END_RUNG
   RUNG wire#w1
      Contact( #Dose_ChiliFresh3.QDOSERun )
      Move(in := #Dose_ChiliFresh3.LastQtyDose, out1 => #Last_Dose_Qty.ChiliFresh3)
   END_RUNG
   RUNG wire#w1
      Contact( #Dose_Garlic.QDOSERun )
      Move(in := #Dose_Garlic.LastQtyDose, out1 => #Last_Dose_Qty.Garlic)
   END_RUNG
   RUNG wire#w1
      Contact( #Dose_HW.QDOSERun )
      Move(in := #"HW Flushing".Qty."Flush to Blend Act", out1 => #Last_Dose_Qty.HW)
   END_RUNG
   RUNG wire#w1
      Contact( #Dose_Vinegar.QDOSERun )
      Move(in := #Dose_Vinegar.LastQtyDose, out1 => #Last_Dose_Qty.Vinegar)
   END_RUNG
   RUNG wire#w1
      Contact( #Dose_Sugar.QDOSERun )
      Move(in := #Dose_Sugar.LastQtyDose, out1 => #Last_Dose_Qty.Sugar)
   END_RUNG
   RUNG wire#w1
      Contact( #Dose_Salt.QDOSERun )
      Move(in := #Dose_Salt.LastQtyDose, out1 => #Last_Dose_Qty.Salt)
   END_RUNG
   RUNG wire#w1
      Contact( #Dose_ProWater.QDOSERun )
      Move(in := #Dose_ProWater.LastQtyDose, out1 => #Last_Dose_Qty.ProWater)
   END_RUNG
   RUNG wire#w1
      Contact( #Dose_Homomixer.QDOSERun )
      Move(in := #Dose_Homomixer.LastQtyDose, out1 => #Last_Dose_Qty.Homomixer)
   END_RUNG
   // the same network as SCL:
   IF #AlwaysON AND #Dose_ChiliAwetan1.QDOSERun THEN
       #Last_Dose_Qty.ChiliAwetan1 := #Dose_ChiliAwetan1.LastQtyDose;
   END_IF;
   IF #AlwaysON AND #Dose_ChiliAwetan2.QDOSERun THEN
       #Last_Dose_Qty.ChiliAwetan2 := #Dose_ChiliAwetan2.LastQtyDose;
   END_IF;
   IF #AlwaysON AND #Dose_ChiliAwetan3.QDOSERun THEN
       #Last_Dose_Qty.ChiliAwetan3 := #Dose_ChiliAwetan3.LastQtyDose;
   END_IF;
   IF #AlwaysON AND #Dose_Tomato.QDOSERun THEN #Last_Dose_Qty.Tomato := #Dose_Tomato.LastQtyDose; END_IF;
   IF #AlwaysON AND #Dose_ChiliFresh1.QDOSERun THEN
       #Last_Dose_Qty.ChiliFresh1 := #Dose_ChiliFresh1.LastQtyDose;
   END_IF;
   IF #AlwaysON AND #Dose_ChiliFresh2.QDOSERun THEN
       #Last_Dose_Qty.ChiliFresh2 := #Dose_ChiliFresh2.LastQtyDose;
   END_IF;
   IF #AlwaysON AND #Dose_ChiliFresh3.QDOSERun THEN
       #Last_Dose_Qty.ChiliFresh3 := #Dose_ChiliFresh3.LastQtyDose;
   END_IF;
   IF #AlwaysON AND #Dose_Garlic.QDOSERun THEN #Last_Dose_Qty.Garlic := #Dose_Garlic.LastQtyDose; END_IF;
   IF #AlwaysON AND #Dose_HW.QDOSERun THEN
       #Last_Dose_Qty.HW := #"HW Flushing".Qty."Flush to Blend Act";
   END_IF;
   IF #AlwaysON AND #Dose_Vinegar.QDOSERun THEN #Last_Dose_Qty.Vinegar := #Dose_Vinegar.LastQtyDose; END_IF;
   IF #AlwaysON AND #Dose_Sugar.QDOSERun THEN #Last_Dose_Qty.Sugar := #Dose_Sugar.LastQtyDose; END_IF;
   IF #AlwaysON AND #Dose_Salt.QDOSERun THEN #Last_Dose_Qty.Salt := #Dose_Salt.LastQtyDose; END_IF;
   IF #AlwaysON AND #Dose_ProWater.QDOSERun THEN
       #Last_Dose_Qty.ProWater := #Dose_ProWater.LastQtyDose;
   END_IF;
   IF #AlwaysON AND #Dose_Homomixer.QDOSERun THEN
       #Last_Dose_Qty.Homomixer := #Dose_Homomixer.LastQtyDose;
   END_IF;
END_REGION

REGION Network 124: Reset Last Dose Qty After CIP Tank
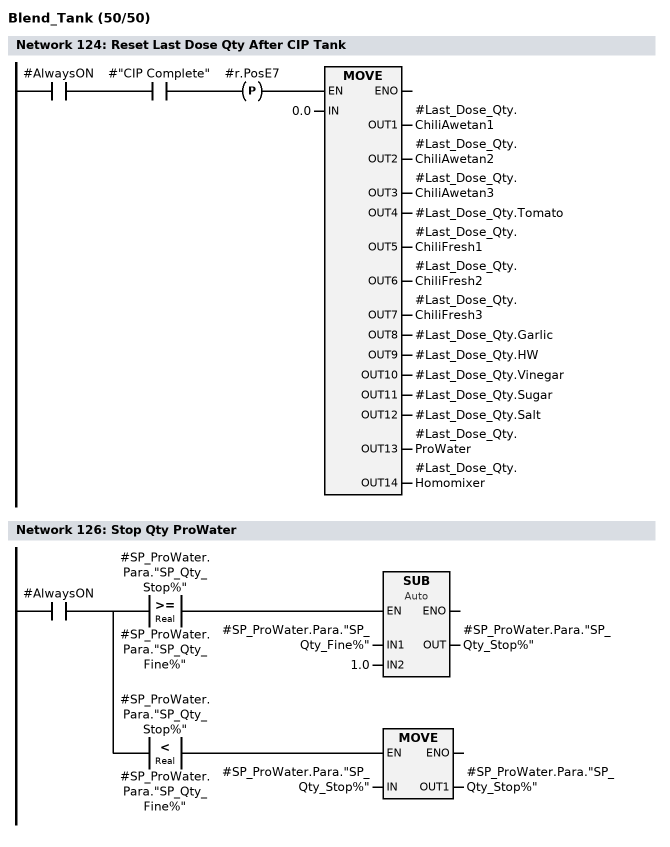
   RUNG wire#powerrail
      Contact( #AlwaysON )
      Contact( #"CIP Complete" )
      P_Trig( #r.PosE7 )
      Move(in := 0.0, out1 => #Last_Dose_Qty.ChiliAwetan1, out2 => #Last_Dose_Qty.ChiliAwetan2, out3 => #Last_Dose_Qty.ChiliAwetan3, out4 => #Last_Dose_Qty.Tomato, out5 => #Last_Dose_Qty.ChiliFresh1, out6 => #Last_Dose_Qty.ChiliFresh2, out7 => #Last_Dose_Qty.ChiliFresh3, out8 => #Last_Dose_Qty.Garlic, out9 => #Last_Dose_Qty.HW, out10 => #Last_Dose_Qty.Vinegar, out11 => #Last_Dose_Qty.Sugar, out12 => #Last_Dose_Qty.Salt, out13 => #Last_Dose_Qty.ProWater, out14 => #Last_Dose_Qty.Homomixer)
   END_RUNG
   // the same network as SCL:
   #_w1 := #AlwaysON AND #"CIP Complete";
   #_w2 := #_w1 AND NOT #r.PosE7;   // rising edge
   #r.PosE7 := #_w1;
   IF #_w2 THEN
       #Last_Dose_Qty.ChiliAwetan1 := 0.0;
       #Last_Dose_Qty.ChiliAwetan2 := 0.0;
       #Last_Dose_Qty.ChiliAwetan3 := 0.0;
       #Last_Dose_Qty.Tomato := 0.0;
       #Last_Dose_Qty.ChiliFresh1 := 0.0;
       #Last_Dose_Qty.ChiliFresh2 := 0.0;
       #Last_Dose_Qty.ChiliFresh3 := 0.0;
       #Last_Dose_Qty.Garlic := 0.0;
       #Last_Dose_Qty.HW := 0.0;
       #Last_Dose_Qty.Vinegar := 0.0;
       #Last_Dose_Qty.Sugar := 0.0;
       #Last_Dose_Qty.Salt := 0.0;
       #Last_Dose_Qty.ProWater := 0.0;
       #Last_Dose_Qty.Homomixer := 0.0;
   END_IF;
END_REGION

REGION Network 126: Stop Qty ProWater
   RUNG wire#powerrail
      Contact( #AlwaysON )
      wire#w1
      { S7_Templates := "SrcType := Real" } GE_Contact(in1 := #SP_ProWater.Para."SP_Qty_Stop%", in2 := #SP_ProWater.Para."SP_Qty_Fine%")
      Sub(in1 := #SP_ProWater.Para."SP_Qty_Fine%", in2 := 1.0, out => #SP_ProWater.Para."SP_Qty_Stop%")
   END_RUNG
   RUNG wire#w1
      { S7_Templates := "SrcType := Real" } LT_Contact(in1 := #SP_ProWater.Para."SP_Qty_Stop%", in2 := #SP_ProWater.Para."SP_Qty_Fine%")
      Move(in := #SP_ProWater.Para."SP_Qty_Stop%", out1 => #SP_ProWater.Para."SP_Qty_Stop%")
   END_RUNG
   // the same network as SCL:
   IF #AlwaysON AND (#SP_ProWater.Para."SP_Qty_Stop%" >= #SP_ProWater.Para."SP_Qty_Fine%") THEN
       #SP_ProWater.Para."SP_Qty_Stop%" := #SP_ProWater.Para."SP_Qty_Fine%" - 1.0;
   END_IF;
   IF #AlwaysON AND (#SP_ProWater.Para."SP_Qty_Stop%" < #SP_ProWater.Para."SP_Qty_Fine%") THEN
       #SP_ProWater.Para."SP_Qty_Stop%" := #SP_ProWater.Para."SP_Qty_Stop%";
   END_IF;
END_REGION
END_FUNCTION_BLOCK

FUNCTION_BLOCK "IO_Valve_Blend20"   // FB24, LAD
{ S7_Optimized_Access := 'FALSE' }
VERSION : 0.1
// stored: AutoNumber true, IsIECCheckEnabled false, SetENOAutomatically false, UDAEnableTagReadback false
   VAR_INPUT
      "lock 1" : Bool;
      "lock 2" : Bool;
      "lock 3" : Bool;
      "lock 4" : Bool;
      init : Bool;
      reset : Bool;
      testing : Bool;
   END_VAR
   VAR
      "AV-20.01" : "Valve";
      "AV-20.02" : "Valve";
      "AV-20.03" : "Valve";
      "AV-20.04" : "Valve";
      "AV-20.05" : "Valve";
      "AV-20.06" : "Valve";
      "AV-20.07" : "Valve";
      "AV-20.08" : "Valve";
      "AV-20.09" : "Valve";
      "AV-20.10" : "Valve";
      "AV-20.11" : "Valve";
      "AV-20.21" : "Valve";
      "AV-20.22" : "Valve";
      "AV-20.23" : "Valve";
      "AV-20.24" : "Valve";
      "AV-20.25" : "Valve";
      "AV-20.26" : "Valve";
      "AV-20.27" : "Valve";
      "AV-20.28" : "Valve";
      "AV-20.29" : "Valve";
      "AV-20.30" : "Valve";
      "AV-20.31" : "Valve";
      "AV-20.32" : "Valve";
      "AV-20.33" : "Valve";
      "AV-20.34" : "Valve";
      "AV-20.35" : "Valve";
      "AV-20.36" : "Valve";
      "AV-20.37" : "Valve";
      "AV-20.41" : "Valve";
      "AV-20.42" : "Valve";
   END_VAR
BEGIN

REGION Network 1 (SCL): FB OPEN AND CLOSE VALVE T-20
   IF #testing THEN
       // Statement section IF
       #"AV-20.01".FB_OPEN := #"AV-20.01".QCMD_OP;
       #"AV-20.01".FB_CLOSE := NOT #"AV-20.01".QCMD_OP;
       #"AV-20.02".FB_OPEN := #"AV-20.02".QCMD_OP;
       #"AV-20.02".FB_CLOSE := NOT #"AV-20.02".QCMD_OP;
       #"AV-20.03".FB_OPEN := #"AV-20.03".QCMD_OP;
       #"AV-20.03".FB_CLOSE := NOT #"AV-20.03".QCMD_OP;
       #"AV-20.04".FB_OPEN := #"AV-20.04".QCMD_OP;
       #"AV-20.04".FB_CLOSE := NOT #"AV-20.04".QCMD_OP;
       #"AV-20.05".FB_OPEN := #"AV-20.05".QCMD_OP;
       #"AV-20.05".FB_CLOSE := NOT #"AV-20.05".QCMD_OP;
       #"AV-20.06".FB_OPEN := #"AV-20.06".QCMD_OP;
       #"AV-20.06".FB_CLOSE := NOT #"AV-20.06".QCMD_OP;
       #"AV-20.07".FB_OPEN := #"AV-20.07".QCMD_OP;
       #"AV-20.07".FB_CLOSE := NOT #"AV-20.07".QCMD_OP;
       #"AV-20.08".FB_OPEN := #"AV-20.08".QCMD_OP;
       #"AV-20.08".FB_CLOSE := NOT #"AV-20.08".QCMD_OP;
       #"AV-20.09".FB_OPEN := #"AV-20.09".QCMD_OP;
       #"AV-20.09".FB_CLOSE := NOT #"AV-20.09".QCMD_OP;
       #"AV-20.10".FB_OPEN := #"AV-20.10".QCMD_OP;
       #"AV-20.10".FB_CLOSE := NOT #"AV-20.10".QCMD_OP;
       #"AV-20.11".FB_OPEN := #"AV-20.11".QCMD_OP;
       #"AV-20.11".FB_CLOSE := NOT #"AV-20.11".QCMD_OP;
       #"AV-20.21".FB_OPEN := #"AV-20.21".QCMD_OP;
       #"AV-20.21".FB_CLOSE := NOT #"AV-20.21".QCMD_OP;
       #"AV-20.22".FB_OPEN := #"AV-20.22".QCMD_OP;
       #"AV-20.22".FB_CLOSE := NOT #"AV-20.22".QCMD_OP;
       #"AV-20.23".FB_OPEN := #"AV-20.23".QCMD_OP;
       #"AV-20.23".FB_CLOSE := NOT #"AV-20.23".QCMD_OP;
       #"AV-20.24".FB_OPEN := #"AV-20.24".QCMD_OP;
       #"AV-20.24".FB_CLOSE := NOT #"AV-20.24".QCMD_OP;
       #"AV-20.25".FB_OPEN := #"AV-20.25".QCMD_OP;
       #"AV-20.25".FB_CLOSE := NOT #"AV-20.25".QCMD_OP;
       #"AV-20.26".FB_OPEN := #"AV-20.26".QCMD_OP;
       #"AV-20.26".FB_CLOSE := NOT #"AV-20.26".QCMD_OP;
       #"AV-20.27".FB_OPEN := #"AV-20.27".QCMD_OP;
       #"AV-20.27".FB_CLOSE := NOT #"AV-20.27".QCMD_OP;
       #"AV-20.28".FB_OPEN := #"AV-20.28".QCMD_OP;
       #"AV-20.28".FB_CLOSE := NOT #"AV-20.28".QCMD_OP;
       #"AV-20.29".FB_OPEN := #"AV-20.29".QCMD_OP;
       #"AV-20.29".FB_CLOSE := NOT #"AV-20.29".QCMD_OP;
       #"AV-20.30".FB_OPEN := #"AV-20.30".QCMD_OP;
       #"AV-20.30".FB_CLOSE := NOT #"AV-20.30".QCMD_OP;
       #"AV-20.31".FB_OPEN := #"AV-20.31".QCMD_OP;
       #"AV-20.31".FB_CLOSE := NOT #"AV-20.31".QCMD_OP;
       #"AV-20.32".FB_OPEN := #"AV-20.32".QCMD_OP;
       #"AV-20.32".FB_CLOSE := NOT #"AV-20.32".QCMD_OP;
       #"AV-20.33".FB_OPEN := #"AV-20.33".QCMD_OP;
       #"AV-20.33".FB_CLOSE := NOT #"AV-20.33".QCMD_OP;
       #"AV-20.34".FB_OPEN := #"AV-20.34".QCMD_OP;
       #"AV-20.34".FB_CLOSE := NOT #"AV-20.34".QCMD_OP;
       #"AV-20.35".FB_OPEN := #"AV-20.35".QCMD_OP;
       #"AV-20.35".FB_CLOSE := NOT #"AV-20.35".QCMD_OP;
       #"AV-20.36".FB_OPEN := #"AV-20.36".QCMD_OP;
       #"AV-20.36".FB_CLOSE := NOT #"AV-20.36".QCMD_OP;
       #"AV-20.37".FB_OPEN := #"AV-20.37".QCMD_OP;
       #"AV-20.37".FB_CLOSE := NOT #"AV-20.37".QCMD_OP;
       #"AV-20.41".FB_OPEN := #"AV-20.41".QCMD_OP;
       #"AV-20.41".FB_CLOSE := NOT #"AV-20.41".QCMD_OP;
       #"AV-20.42".FB_OPEN := #"AV-20.42".QCMD_OP;
       #"AV-20.42".FB_CLOSE := NOT #"AV-20.42".QCMD_OP;
   ELSE
       // Statement section ELSE
       #"AV-20.01".FB_OPEN := #"AV-20.01".QCMD_OP;
       #"AV-20.01".FB_CLOSE := NOT #"AV-20.01".QCMD_OP;
       #"AV-20.02".FB_OPEN := NOT "ZSC-20.02";
       #"AV-20.02".FB_CLOSE := "ZSC-20.02";
       #"AV-20.03".FB_OPEN := NOT "ZSC-20.03";
       #"AV-20.03".FB_CLOSE := "ZSC-20.03";
       #"AV-20.04".FB_OPEN := #"AV-20.04".QCMD_OP;
       #"AV-20.04".FB_CLOSE := NOT #"AV-20.04".QCMD_OP;
       #"AV-20.05".FB_OPEN := NOT "ZSC-20.05";
       #"AV-20.05".FB_CLOSE := "ZSC-20.05";
       #"AV-20.06".FB_OPEN := NOT "ZSC-20.06";
       #"AV-20.06".FB_CLOSE := "ZSC-20.06";
       #"AV-20.07".FB_OPEN := #"AV-20.07".QCMD_OP;
       #"AV-20.07".FB_CLOSE := NOT #"AV-20.07".QCMD_OP;
       #"AV-20.08".FB_OPEN := NOT "ZSC-20.08";
       #"AV-20.08".FB_CLOSE := "ZSC-20.08";
       #"AV-20.09".FB_OPEN := NOT "ZSC-20.09";
       #"AV-20.09".FB_CLOSE := "ZSC-20.09";
       #"AV-20.10".FB_OPEN := #"AV-20.10".QCMD_OP;
       #"AV-20.10".FB_CLOSE := NOT #"AV-20.10".QCMD_OP;
       #"AV-20.11".FB_OPEN := NOT "ZSC-20.11";
       #"AV-20.11".FB_CLOSE := "ZSC-20.11";
       #"AV-20.21".FB_OPEN := NOT "ZSC-20.21";
       #"AV-20.21".FB_CLOSE := "ZSC-20.21";
       #"AV-20.22".FB_OPEN := #"AV-20.22".QCMD_OP;
       #"AV-20.22".FB_CLOSE := NOT #"AV-20.22".QCMD_OP;
       #"AV-20.23".FB_OPEN := NOT "ZSC-20.23";
       #"AV-20.23".FB_CLOSE := "ZSC-20.23";
       #"AV-20.24".FB_OPEN := NOT "ZSC-20.24";
       #"AV-20.24".FB_CLOSE := "ZSC-20.24";
       #"AV-20.25".FB_OPEN := NOT "ZSC-20.25";
       #"AV-20.25".FB_CLOSE := "ZSC-20.25";
       #"AV-20.26".FB_OPEN := #"AV-20.26".QCMD_OP;
       #"AV-20.26".FB_CLOSE := NOT #"AV-20.26".QCMD_OP;
       #"AV-20.27".FB_OPEN := NOT "ZSC-20.27";
       #"AV-20.27".FB_CLOSE := "ZSC-20.27";
       #"AV-20.28".FB_OPEN := NOT "ZSC-20.28";
       #"AV-20.28".FB_CLOSE := "ZSC-20.28";
       #"AV-20.29".FB_OPEN := #"AV-20.29".QCMD_OP;
       #"AV-20.29".FB_CLOSE := NOT #"AV-20.29".QCMD_OP;
       #"AV-20.30".FB_OPEN := #"AV-20.30".QCMD_OP;
       #"AV-20.30".FB_CLOSE := NOT #"AV-20.30".QCMD_OP;
       #"AV-20.31".FB_OPEN := NOT "ZSC-20.31";
       #"AV-20.31".FB_CLOSE := "ZSC-20.31";
       #"AV-20.32".FB_OPEN := NOT "ZSC-20.32";
       #"AV-20.32".FB_CLOSE := "ZSC-20.32";
       #"AV-20.33".FB_OPEN := NOT "ZSC-20.33";
       #"AV-20.33".FB_CLOSE := "ZSC-20.33";
       #"AV-20.34".FB_OPEN := NOT "ZSC-20.34";
       #"AV-20.34".FB_CLOSE := "ZSC-20.34";
       #"AV-20.35".FB_OPEN := NOT "ZSC-20.35";
       #"AV-20.35".FB_CLOSE := "ZSC-20.35";
       #"AV-20.36".FB_OPEN := NOT "ZSC-20.36";
       #"AV-20.36".FB_CLOSE := "ZSC-20.36";
       #"AV-20.37".FB_OPEN := NOT "ZSC-20.37";
       #"AV-20.37".FB_CLOSE := "ZSC-20.37";
       #"AV-20.41".FB_OPEN := #"AV-20.41".QCMD_OP;
       #"AV-20.41".FB_CLOSE := NOT #"AV-20.41".QCMD_OP;
       #"AV-20.42".FB_OPEN := #"AV-20.42".QCMD_OP;
       #"AV-20.42".FB_CLOSE := NOT #"AV-20.42".QCMD_OP;
   END_IF;
END_REGION

NETWORK
TITLE = FB MONITORING TIME VALVE T-20
// FB OPEN TIME
      L     T#20s;
      T     #"AV-20.01".MON_T;
      T     #"AV-20.02".MON_T;
      T     #"AV-20.03".MON_T;
      T     #"AV-20.04".MON_T;
      T     #"AV-20.05".MON_T;
      T     #"AV-20.06".MON_T;
      T     #"AV-20.07".MON_T;
      T     #"AV-20.08".MON_T;
      T     #"AV-20.09".MON_T;
      T     #"AV-20.10".MON_T;
      T     #"AV-20.11".MON_T;
      T     #"AV-20.21".MON_T;
      T     #"AV-20.22".MON_T;
      T     #"AV-20.23".MON_T;
      T     #"AV-20.24".MON_T;
      T     #"AV-20.25".MON_T;
      T     #"AV-20.26".MON_T;
      T     #"AV-20.27".MON_T;
      T     #"AV-20.28".MON_T;
      T     #"AV-20.29".MON_T;
      T     #"AV-20.30".MON_T;
      T     #"AV-20.31".MON_T;
      T     #"AV-20.32".MON_T;
      T     #"AV-20.33".MON_T;
      T     #"AV-20.34".MON_T;
      T     #"AV-20.35".MON_T;
      T     #"AV-20.36".MON_T;
      T     #"AV-20.37".MON_T;
      T     #"AV-20.41".MON_T;
      T     #"AV-20.42".MON_T;

// FB CLOSE TIME
      L     T#20s;
      T     #"AV-20.01".MON_T_CLOSE;
      T     #"AV-20.02".MON_T_CLOSE;
      T     #"AV-20.03".MON_T_CLOSE;
      T     #"AV-20.04".MON_T_CLOSE;
      T     #"AV-20.05".MON_T_CLOSE;
      T     #"AV-20.06".MON_T_CLOSE;
      T     #"AV-20.07".MON_T_CLOSE;
      T     #"AV-20.08".MON_T_CLOSE;
      T     #"AV-20.09".MON_T_CLOSE;
      T     #"AV-20.10".MON_T_CLOSE;
      T     #"AV-20.11".MON_T_CLOSE;
      T     #"AV-20.21".MON_T_CLOSE;
      T     #"AV-20.22".MON_T_CLOSE;
      T     #"AV-20.23".MON_T_CLOSE;
      T     #"AV-20.24".MON_T_CLOSE;
      T     #"AV-20.25".MON_T_CLOSE;
      T     #"AV-20.26".MON_T_CLOSE;
      T     #"AV-20.27".MON_T_CLOSE;
      T     #"AV-20.28".MON_T_CLOSE;
      T     #"AV-20.29".MON_T_CLOSE;
      T     #"AV-20.30".MON_T_CLOSE;
      T     #"AV-20.31".MON_T_CLOSE;
      T     #"AV-20.32".MON_T_CLOSE;
      T     #"AV-20.33".MON_T_CLOSE;
      T     #"AV-20.34".MON_T_CLOSE;
      T     #"AV-20.35".MON_T_CLOSE;
      T     #"AV-20.36".MON_T_CLOSE;
      T     #"AV-20.37".MON_T_CLOSE;
      T     #"AV-20.41".MON_T_CLOSE;
      T     #"AV-20.42".MON_T_CLOSE;


REGION Network 3: AV-20.01
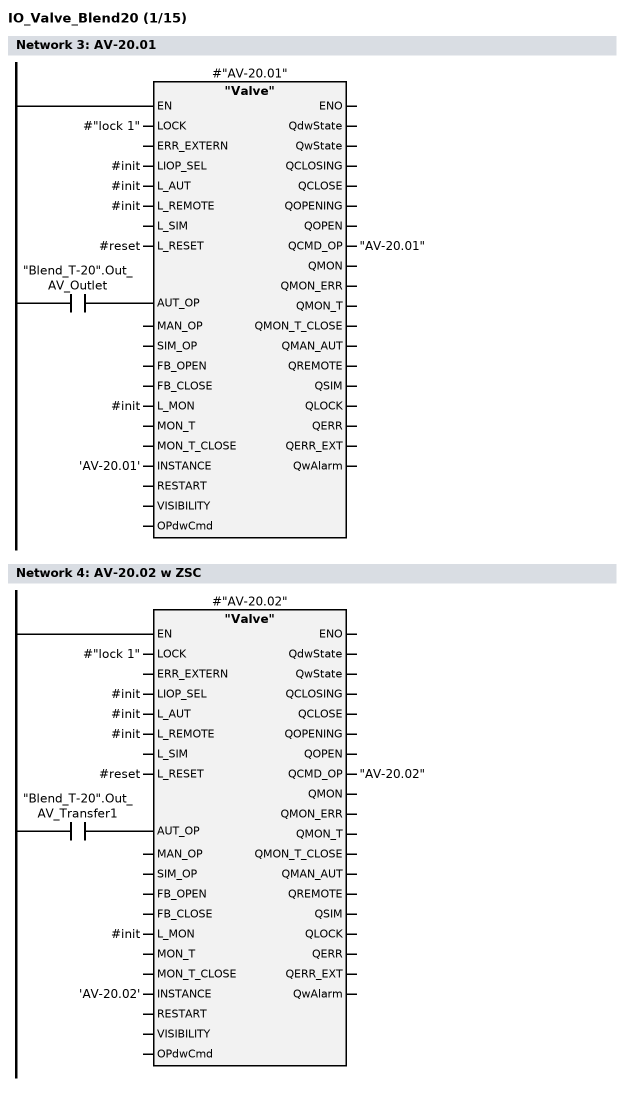
   RUNG wire#powerrail
      #"AV-20.01"(AUT_OP := wire#w1, LOCK := #"lock 1", ERR_EXTERN :=, LIOP_SEL := #init, L_AUT := #init, L_REMOTE := #init, L_SIM :=, L_RESET := #reset, MAN_OP :=, SIM_OP :=, FB_OPEN :=, FB_CLOSE :=, L_MON := #init, MON_T :=, MON_T_CLOSE :=, INSTANCE := 'AV-20.01', RESTART :=, VISIBILITY :=, OPdwCmd :=, QdwState =>, QwState =>, QCLOSING =>, QCLOSE =>, QOPENING =>, QOPEN =>, QCMD_OP => "AV-20.01", QMON =>, QMON_ERR =>, QMON_T =>, QMON_T_CLOSE =>, QMAN_AUT =>, QREMOTE =>, QSIM =>, QLOCK =>, QERR =>, QERR_EXT =>, QwAlarm =>)
   END_RUNG
   RUNG wire#powerrail
      Contact( "Blend_T-20".Out_AV_Outlet )
   END_RUNG wire#w1
   // the same network as SCL:
   #"AV-20.01"(LOCK := #"lock 1",   // "Valve"
               LIOP_SEL := #init,
               L_AUT := #init,
               L_REMOTE := #init,
               L_RESET := #reset,
               AUT_OP := "Blend_T-20".Out_AV_Outlet,
               L_MON := #init,
               INSTANCE := 'AV-20.01',
               QCMD_OP => "AV-20.01");
END_REGION

REGION Network 4: AV-20.02 w ZSC
   RUNG wire#powerrail
      #"AV-20.02"(AUT_OP := wire#w1, LOCK := #"lock 1", ERR_EXTERN :=, LIOP_SEL := #init, L_AUT := #init, L_REMOTE := #init, L_SIM :=, L_RESET := #reset, MAN_OP :=, SIM_OP :=, FB_OPEN :=, FB_CLOSE :=, L_MON := #init, MON_T :=, MON_T_CLOSE :=, INSTANCE := 'AV-20.02', RESTART :=, VISIBILITY :=, OPdwCmd :=, QdwState =>, QwState =>, QCLOSING =>, QCLOSE =>, QOPENING =>, QOPEN =>, QCMD_OP => "AV-20.02", QMON =>, QMON_ERR =>, QMON_T =>, QMON_T_CLOSE =>, QMAN_AUT =>, QREMOTE =>, QSIM =>, QLOCK =>, QERR =>, QERR_EXT =>, QwAlarm =>)
   END_RUNG
   RUNG wire#powerrail
      Contact( "Blend_T-20".Out_AV_Transfer1 )
   END_RUNG wire#w1
   // the same network as SCL:
   #"AV-20.02"(LOCK := #"lock 1",   // "Valve"
               LIOP_SEL := #init,
               L_AUT := #init,
               L_REMOTE := #init,
               L_RESET := #reset,
               AUT_OP := "Blend_T-20".Out_AV_Transfer1,
               L_MON := #init,
               INSTANCE := 'AV-20.02',
               QCMD_OP => "AV-20.02");
END_REGION

REGION Network 5: AV-20.03 w ZSC
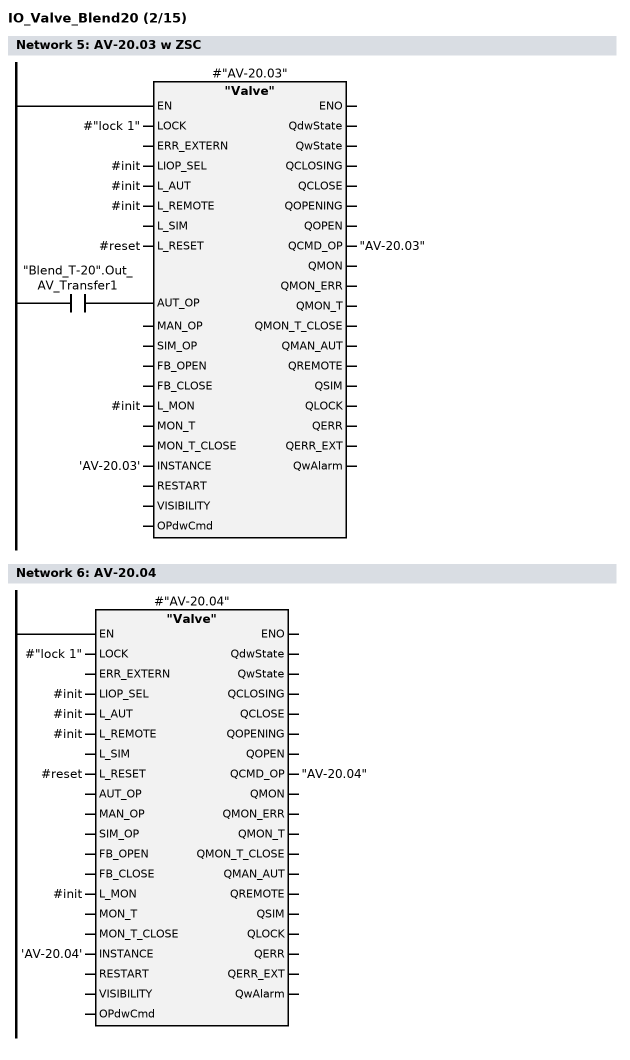
   RUNG wire#powerrail
      #"AV-20.03"(AUT_OP := wire#w1, LOCK := #"lock 1", ERR_EXTERN :=, LIOP_SEL := #init, L_AUT := #init, L_REMOTE := #init, L_SIM :=, L_RESET := #reset, MAN_OP :=, SIM_OP :=, FB_OPEN :=, FB_CLOSE :=, L_MON := #init, MON_T :=, MON_T_CLOSE :=, INSTANCE := 'AV-20.03', RESTART :=, VISIBILITY :=, OPdwCmd :=, QdwState =>, QwState =>, QCLOSING =>, QCLOSE =>, QOPENING =>, QOPEN =>, QCMD_OP => "AV-20.03", QMON =>, QMON_ERR =>, QMON_T =>, QMON_T_CLOSE =>, QMAN_AUT =>, QREMOTE =>, QSIM =>, QLOCK =>, QERR =>, QERR_EXT =>, QwAlarm =>)
   END_RUNG
   RUNG wire#powerrail
      Contact( "Blend_T-20".Out_AV_Transfer1 )
   END_RUNG wire#w1
   // the same network as SCL:
   #"AV-20.03"(LOCK := #"lock 1",   // "Valve"
               LIOP_SEL := #init,
               L_AUT := #init,
               L_REMOTE := #init,
               L_RESET := #reset,
               AUT_OP := "Blend_T-20".Out_AV_Transfer1,
               L_MON := #init,
               INSTANCE := 'AV-20.03',
               QCMD_OP => "AV-20.03");
END_REGION

REGION Network 6: AV-20.04
   RUNG wire#powerrail
      #"AV-20.04"(LOCK := #"lock 1", ERR_EXTERN :=, LIOP_SEL := #init, L_AUT := #init, L_REMOTE := #init, L_SIM :=, L_RESET := #reset, AUT_OP :=, MAN_OP :=, SIM_OP :=, FB_OPEN :=, FB_CLOSE :=, L_MON := #init, MON_T :=, MON_T_CLOSE :=, INSTANCE := 'AV-20.04', RESTART :=, VISIBILITY :=, OPdwCmd :=, QdwState =>, QwState =>, QCLOSING =>, QCLOSE =>, QOPENING =>, QOPEN =>, QCMD_OP => "AV-20.04", QMON =>, QMON_ERR =>, QMON_T =>, QMON_T_CLOSE =>, QMAN_AUT =>, QREMOTE =>, QSIM =>, QLOCK =>, QERR =>, QERR_EXT =>, QwAlarm =>)
   END_RUNG
   // the same network as SCL:
   #"AV-20.04"(LOCK := #"lock 1",   // "Valve"
               LIOP_SEL := #init,
               L_AUT := #init,
               L_REMOTE := #init,
               L_RESET := #reset,
               L_MON := #init,
               INSTANCE := 'AV-20.04',
               QCMD_OP => "AV-20.04");
END_REGION

REGION Network 7: AV-20.05 w ZSC
